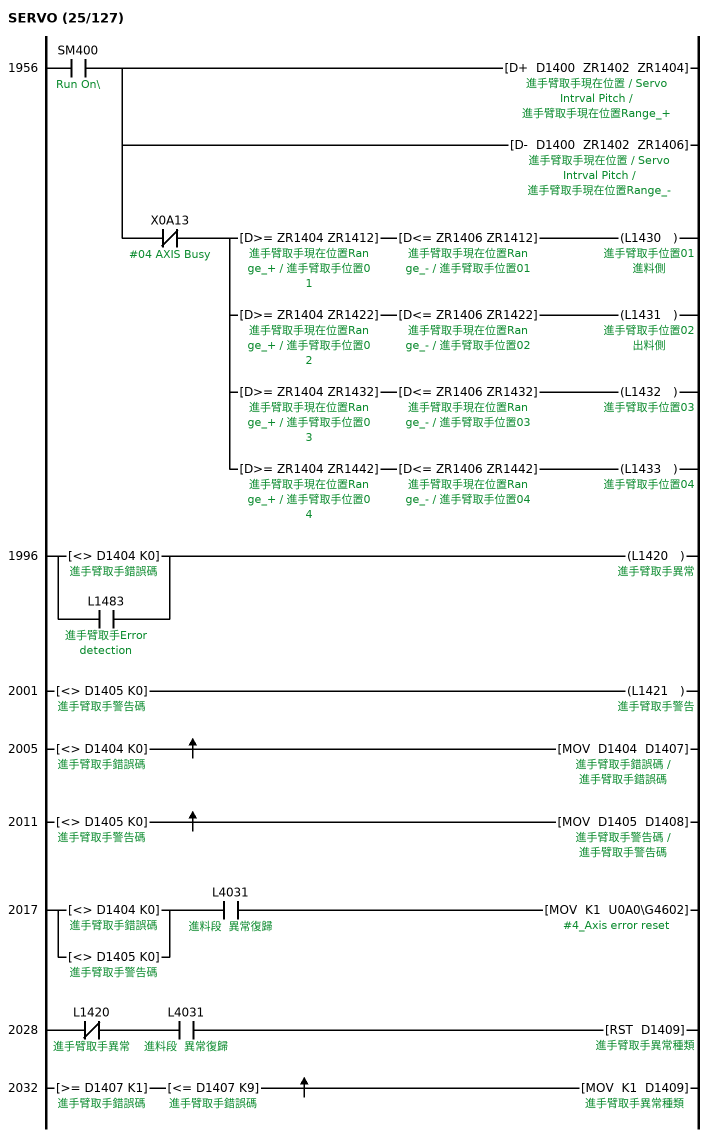
[picture p24: ladder of SERVO, rungs at steps 1956 to 2032]
1956  LD      SM400  ; Run On\
      D+      D1400 ZR1402 ZR1404  ; 進手臂取手現在位置Range_+
      D-      D1400 ZR1402 ZR1406  ; 進手臂取手現在位置Range_-
      ANI     X0A13  ; #04 AXIS Busy
      MPS
      ANDD>=  ZR1404 ZR1412  ; 進手臂取手現在位置Range_+ / 進手臂取手位置01
      ANDD<=  ZR1406 ZR1412  ; 進手臂取手現在位置Range_- / 進手臂取手位置01
      OUT     L1430  ; 進手臂取手位置01  進料側
      MRD
      ANDD>=  ZR1404 ZR1422  ; 進手臂取手現在位置Range_+ / 進手臂取手位置02
      ANDD<=  ZR1406 ZR1422  ; 進手臂取手現在位置Range_- / 進手臂取手位置02
      OUT     L1431  ; 進手臂取手位置02  出料側
      MRD
      ANDD>=  ZR1404 ZR1432  ; 進手臂取手現在位置Range_+ / 進手臂取手位置03
      ANDD<=  ZR1406 ZR1432  ; 進手臂取手現在位置Range_- / 進手臂取手位置03
      OUT     L1432  ; 進手臂取手位置03
      MPP
      ANDD>=  ZR1404 ZR1442  ; 進手臂取手現在位置Range_+ / 進手臂取手位置04
      ANDD<=  ZR1406 ZR1442  ; 進手臂取手現在位置Range_- / 進手臂取手位置04
      OUT     L1433  ; 進手臂取手位置04
1996  LD<>    D1404 K0  ; 進手臂取手錯誤碼
      OR      L1483  ; 進手臂取手Error detection
      OUT     L1420  ; 進手臂取手異常
2001  LD<>    D1405 K0  ; 進手臂取手警告碼
      OUT     L1421  ; 進手臂取手警告
2005  LD<>    D1404 K0  ; 進手臂取手錯誤碼
      MEP
      MOV     D1404 D1407  ; 進手臂取手錯誤碼
2011  LD<>    D1405 K0  ; 進手臂取手警告碼
      MEP
      MOV     D1405 D1408  ; 進手臂取手警告碼
2017  LD<>    D1404 K0  ; 進手臂取手錯誤碼
      OR<>    D1405 K0  ; 進手臂取手警告碼
      AND     L4031  ; 進料段  異常復歸
      MOV     K1 U0A0\G4602  ; #4_Axis error reset
2028  LDI     L1420  ; 進手臂取手異常
      AND     L4031  ; 進料段  異常復歸
      RST     D1409  ; 進手臂取手異常種類
2032  LD>=    D1407 K1  ; 進手臂取手錯誤碼
      AND<=   D1407 K9  ; 進手臂取手錯誤碼
      MEP
      MOV     K1 D1409
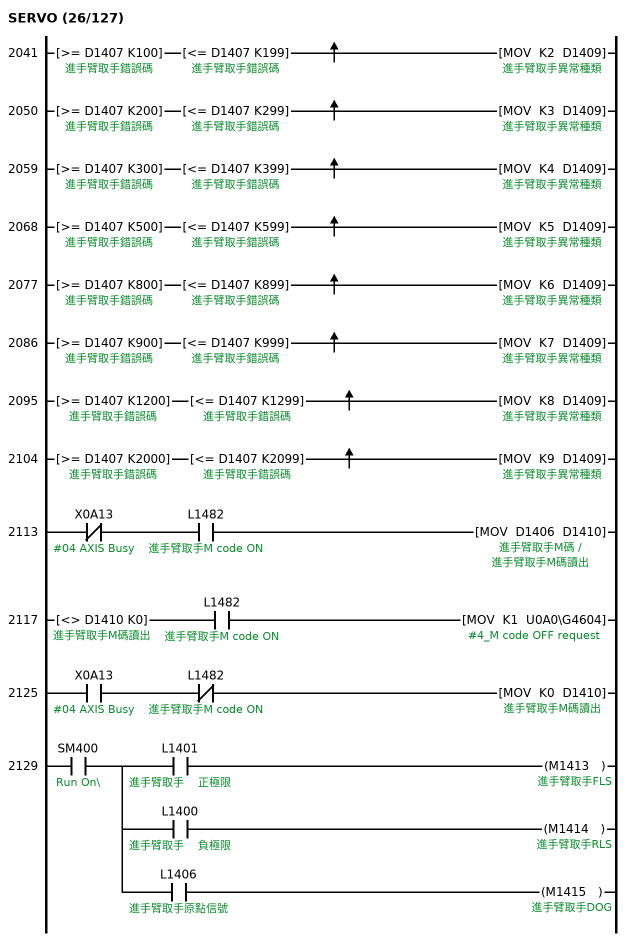
2041  LD>=    D1407 K100  ; 進手臂取手錯誤碼
      AND<=   D1407 K199  ; 進手臂取手錯誤碼
      MEP
      MOV     K2 D1409
2050  LD>=    D1407 K200  ; 進手臂取手錯誤碼
      AND<=   D1407 K299  ; 進手臂取手錯誤碼
      MEP
      MOV     K3 D1409
2059  LD>=    D1407 K300  ; 進手臂取手錯誤碼
      AND<=   D1407 K399  ; 進手臂取手錯誤碼
      MEP
      MOV     K4 D1409
2068  LD>=    D1407 K500  ; 進手臂取手錯誤碼
      AND<=   D1407 K599  ; 進手臂取手錯誤碼
      MEP
      MOV     K5 D1409
2077  LD>=    D1407 K800  ; 進手臂取手錯誤碼
      AND<=   D1407 K899  ; 進手臂取手錯誤碼
      MEP
      MOV     K6 D1409
2086  LD>=    D1407 K900  ; 進手臂取手錯誤碼
      AND<=   D1407 K999  ; 進手臂取手錯誤碼
      MEP
      MOV     K7 D1409
2095  LD>=    D1407 K1200  ; 進手臂取手錯誤碼
      AND<=   D1407 K1299  ; 進手臂取手錯誤碼
      MEP
      MOV     K8 D1409
2104  LD>=    D1407 K2000  ; 進手臂取手錯誤碼
      AND<=   D1407 K2099  ; 進手臂取手錯誤碼
      MEP
      MOV     K9 D1409
2113  LDI     X0A13  ; #04 AXIS Busy
      AND     L1482  ; 進手臂取手M code ON
      MOV     D1406 D1410  ; 進手臂取手M碼讀出
2117  LD<>    D1410 K0  ; 進手臂取手M碼讀出
      AND     L1482  ; 進手臂取手M code ON
      MOV     K1 U0A0\G4604  ; #4_M code OFF request
2125  LD      X0A13  ; #04 AXIS Busy
      ANI     L1482  ; 進手臂取手M code ON
      MOV     K0 D1410
2129  LD      SM400  ; Run On\
      MPS
      AND     L1401  ; 進手臂取手    正極限
      OUT     M1413  ; 進手臂取手FLS
      MRD
      AND     L1400  ; 進手臂取手    負極限
      OUT     M1414  ; 進手臂取手RLS
      MPP
      AND     L1406  ; 進手臂取手原點信號
      OUT     M1415  ; 進手臂取手DOG
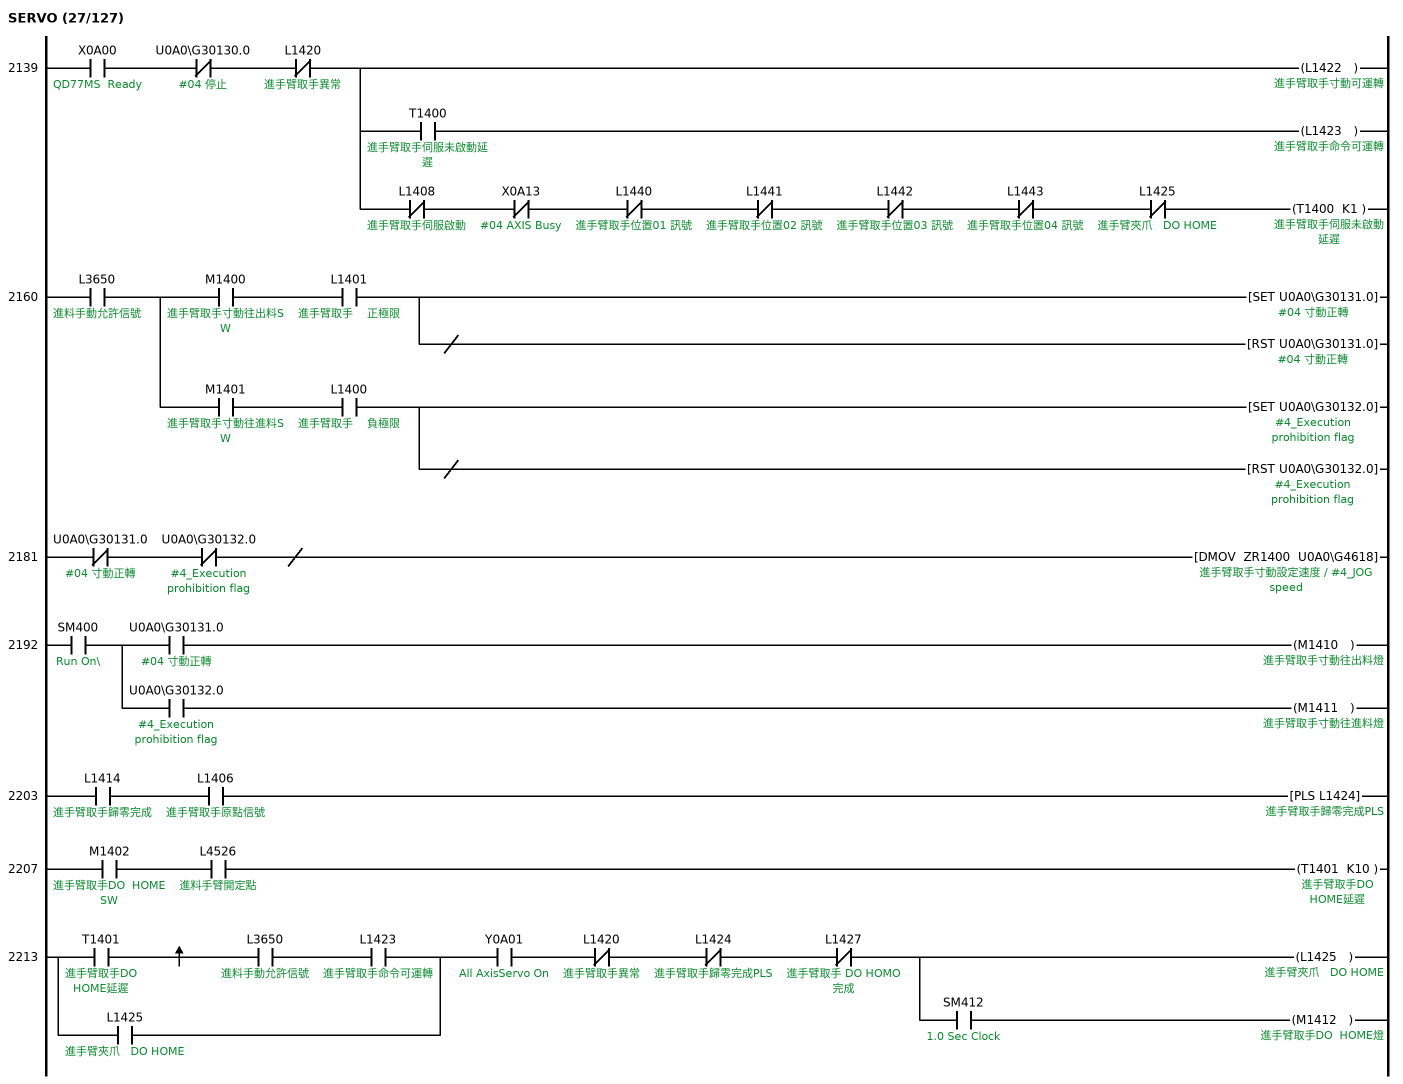
2139  LD      X0A00  ; QD77MS  Ready
      ANI     U0A0\G30130.0  ; #04 停止
      ANI     L1420  ; 進手臂取手異常
      OUT     L1422  ; 進手臂取手寸動可運轉
      MPS
      AND     T1400  ; 進手臂取手伺服未啟動延遲
      OUT     L1423  ; 進手臂取手命令可運轉
      MPP
      ANI     L1408  ; 進手臂取手伺服啟動
      ANI     X0A13  ; #04 AXIS Busy
      ANI     L1440  ; 進手臂取手位置01 訊號
      ANI     L1441  ; 進手臂取手位置02 訊號
      ANI     L1442  ; 進手臂取手位置03 訊號
      ANI     L1443  ; 進手臂取手位置04 訊號
      ANI     L1425  ; 進手臂夾爪   DO HOME
      OUT     T1400 K1  ; 進手臂取手伺服未啟動延遲
2160  LD      L3650  ; 進料手動允許信號
      MPS
      AND     M1400  ; 進手臂取手寸動往出料SW
      AND     L1401  ; 進手臂取手    正極限
      SET     U0A0\G30131.0  ; #04 寸動正轉
      INV
      RST     U0A0\G30131.0  ; #04 寸動正轉
      MPP
      AND     M1401  ; 進手臂取手寸動往進料SW
      AND     L1400  ; 進手臂取手    負極限
      SET     U0A0\G30132.0  ; #4_Execution prohibition flag
      INV
      RST     U0A0\G30132.0  ; #4_Execution prohibition flag
2181  LDI     U0A0\G30131.0  ; #04 寸動正轉
      ANI     U0A0\G30132.0  ; #4_Execution prohibition flag
      INV
      DMOV    ZR1400 U0A0\G4618  ; 進手臂取手寸動設定速度 / #4_JOG     speed
2192  LD      SM400  ; Run On\
      MPS
      AND     U0A0\G30131.0  ; #04 寸動正轉
      OUT     M1410  ; 進手臂取手寸動往出料燈
      MPP
      AND     U0A0\G30132.0  ; #4_Execution prohibition flag
      OUT     M1411  ; 進手臂取手寸動往進料燈
2203  LD      L1414  ; 進手臂取手歸零完成
      AND     L1406  ; 進手臂取手原點信號
      PLS     L1424  ; 進手臂取手歸零完成PLS
2207  LD      M1402  ; 進手臂取手DO  HOME SW
      AND     L4526  ; 進料手臂開定點
      OUT     T1401 K10  ; 進手臂取手DO HOME延遲
2213  LD      T1401  ; 進手臂取手DO HOME延遲
      MEP
      AND     L3650  ; 進料手動允許信號
      AND     L1423  ; 進手臂取手命令可運轉
      OR      L1425  ; 進手臂夾爪   DO HOME
      AND     Y0A01  ; All AxisServo On
      ANI     L1420  ; 進手臂取手異常
      ANI     L1424  ; 進手臂取手歸零完成PLS
      ANI     L1427  ; 進手臂取手 DO HOMO 完成
      OUT     L1425  ; 進手臂夾爪   DO HOME
      AND     SM412  ; 1.0 Sec Clock
      OUT     M1412  ; 進手臂取手DO  HOME燈
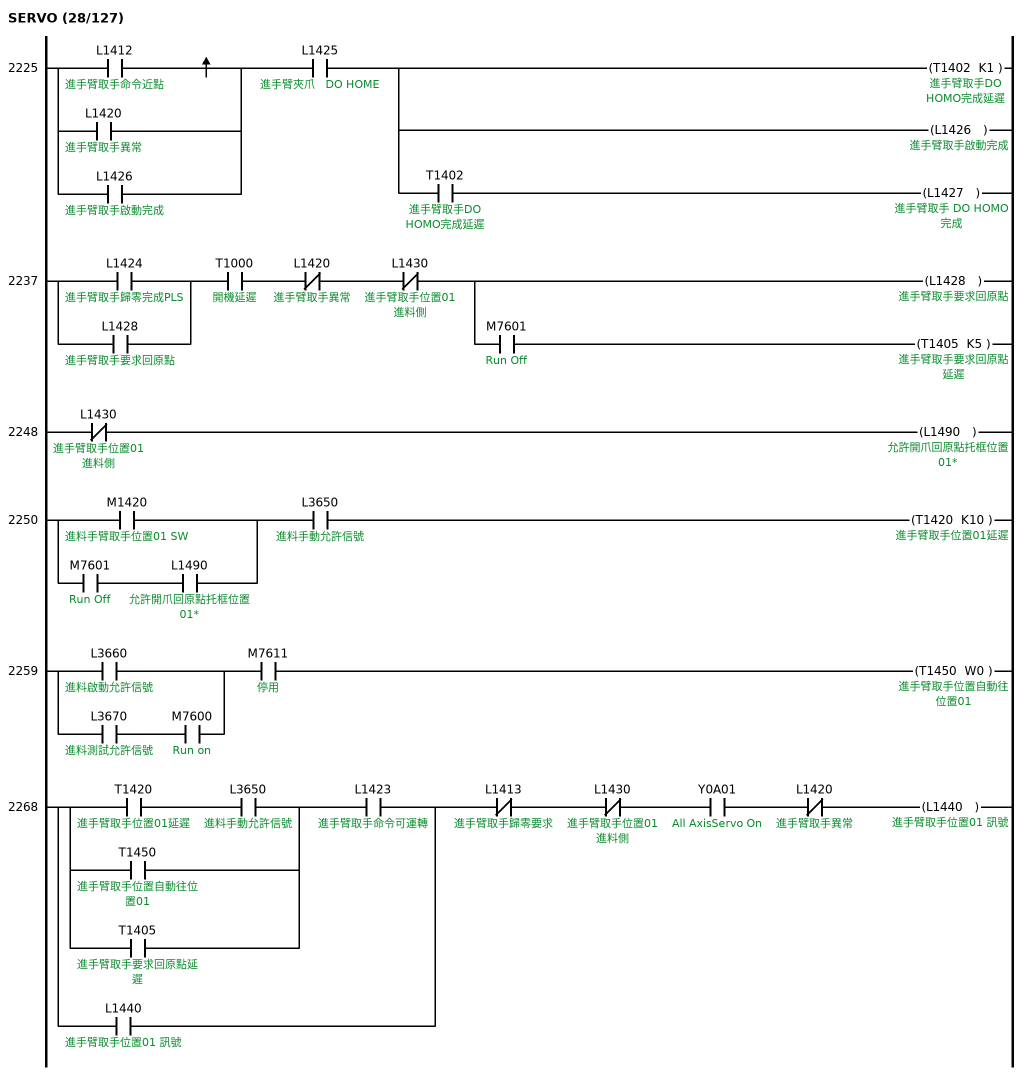
2225  LD      L1412  ; 進手臂取手命令近點
      MEP
      OR      L1420  ; 進手臂取手異常
      OR      L1426  ; 進手臂取手啟動完成
      AND     L1425  ; 進手臂夾爪   DO HOME
      OUT     T1402 K1  ; 進手臂取手DO HOMO完成延遲
      OUT     L1426  ; 進手臂取手啟動完成
      AND     T1402  ; 進手臂取手DO HOMO完成延遲
      OUT     L1427  ; 進手臂取手 DO HOMO 完成
2237  LD      L1424  ; 進手臂取手歸零完成PLS
      OR      L1428  ; 進手臂取手要求回原點
      AND     T1000  ; 開機延遲
      ANI     L1420  ; 進手臂取手異常
      ANI     L1430  ; 進手臂取手位置01  進料側
      OUT     L1428  ; 進手臂取手要求回原點
      AND     M7601  ; Run Off
      OUT     T1405 K5  ; 進手臂取手要求回原點延遲
2248  LDI     L1430  ; 進手臂取手位置01  進料側
      OUT     L1490  ; 允許開爪回原點托框位置01*
2250  LD      M1420  ; 進料手臂取手位置01 SW
      LD      M7601  ; Run Off
      AND     L1490  ; 允許開爪回原點托框位置01*
      ORB
      AND     L3650  ; 進料手動允許信號
      OUT     T1420 K10  ; 進手臂取手位置01延遲
2259  LD      L3660  ; 進料啟動允許信號
      LD      L3670  ; 進料測試允許信號
      AND     M7600  ; Run on
      ORB
      AND     M7611  ; 停用
      OUT     T1450 W0  ; 進手臂取手位置自動往位置01
2268  LD      T1420  ; 進手臂取手位置01延遲
      AND     L3650  ; 進料手動允許信號
      OR      T1450  ; 進手臂取手位置自動往位置01
      OR      T1405  ; 進手臂取手要求回原點延遲
      AND     L1423  ; 進手臂取手命令可運轉
      OR      L1440  ; 進手臂取手位置01 訊號
      ANI     L1413  ; 進手臂取手歸零要求
      ANI     L1430  ; 進手臂取手位置01  進料側
      AND     Y0A01  ; All AxisServo On
      ANI     L1420  ; 進手臂取手異常
      OUT     L1440  ; 進手臂取手位置01 訊號
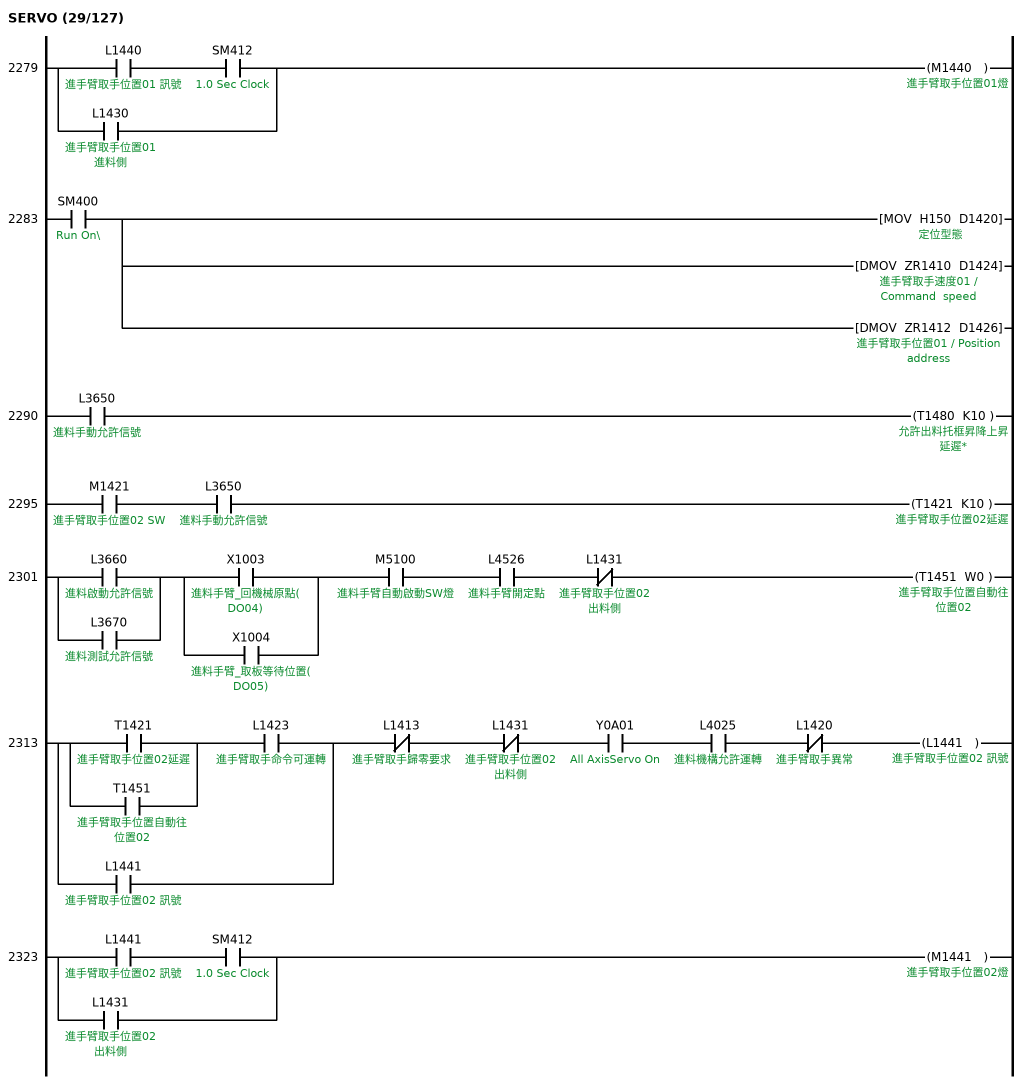
2279  LD      L1440  ; 進手臂取手位置01 訊號
      AND     SM412  ; 1.0 Sec Clock
      OR      L1430  ; 進手臂取手位置01  進料側
      OUT     M1440  ; 進手臂取手位置01燈
2283  LD      SM400  ; Run On\
      MOV     H150 D1420  ; 定位型態
      DMOV    ZR1410 D1424  ; 進手臂取手速度01 / Command  speed
      DMOV    ZR1412 D1426  ; Position address
2290  LD      L3650  ; 進料手動允許信號
      OUT     T1480 K10  ; 允許出料托框昇降上昇延遲*
2295  LD      M1421  ; 進手臂取手位置02 SW
      AND     L3650  ; 進料手動允許信號
      OUT     T1421 K10  ; 進手臂取手位置02延遲
2301  LD      L3660  ; 進料啟動允許信號
      OR      L3670  ; 進料測試允許信號
      LD      X1003  ; 進料手臂_回機械原點(DO04)
      OR      X1004  ; 進料手臂_取板等待位置(DO05)
      ANB
      AND     M5100  ; 進料手臂自動啟動SW燈
      AND     L4526  ; 進料手臂開定點
      ANI     L1431  ; 進手臂取手位置02  出料側
      OUT     T1451 W0  ; 進手臂取手位置自動往  位置02
2313  LD      T1421  ; 進手臂取手位置02延遲
      OR      T1451  ; 進手臂取手位置自動往  位置02
      AND     L1423  ; 進手臂取手命令可運轉
      OR      L1441  ; 進手臂取手位置02 訊號
      ANI     L1413  ; 進手臂取手歸零要求
      ANI     L1431  ; 進手臂取手位置02  出料側
      AND     Y0A01  ; All AxisServo On
      AND     L4025  ; 進料機構允許運轉
      ANI     L1420  ; 進手臂取手異常
      OUT     L1441  ; 進手臂取手位置02 訊號
2323  LD      L1441  ; 進手臂取手位置02 訊號
      AND     SM412  ; 1.0 Sec Clock
      OR      L1431  ; 進手臂取手位置02  出料側
      OUT     M1441  ; 進手臂取手位置02燈
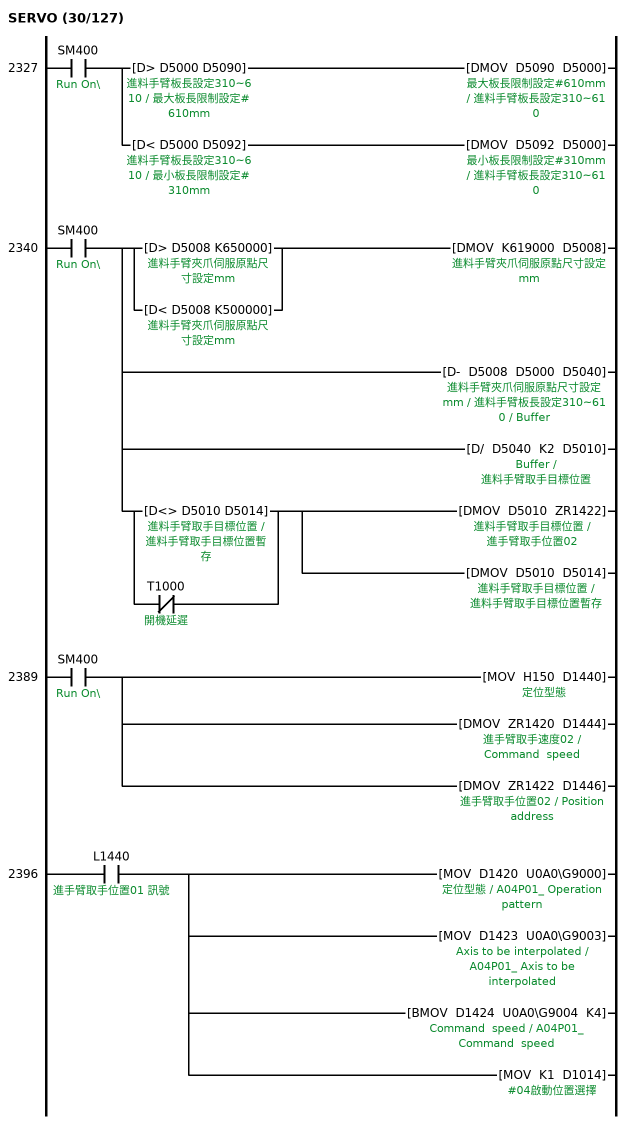
2327  LD      SM400  ; Run On\
      MPS
      ANDD>   D5000 D5090  ; 進料手臂板長設定310~610 / 最大板長限制設定#610mm
      DMOV    D5090 D5000
      MPP
      ANDD<   D5000 D5092  ; 進料手臂板長設定310~610 / 最小板長限制設定#310mm
      DMOV    D5092 D5000
2340  LD      SM400  ; Run On\
      MPS
      LDD>    D5008 K650000  ; 進料手臂夾爪伺服原點尺寸設定mm
      ORD<    D5008 K500000  ; 進料手臂夾爪伺服原點尺寸設定mm
      ANB
      DMOV    K619000 D5008
        [note] /* 手臂夾爪伺服原點尺寸_619mm */
      MPP
      D-      D5008 D5000 D5040
      D/      D5040 K2 D5010  ; 進料手臂取手目標位置
      LDD<>   D5010 D5014  ; 進料手臂取手目標位置 / 進料手臂取手目標位置暫存
      ORI     T1000  ; 開機延遲
      ANB
      DMOV    D5010 ZR1422
      DMOV    D5010 D5014
2389  LD      SM400  ; Run On\
      MOV     H150 D1440  ; 定位型態
      DMOV    ZR1420 D1444  ; 進手臂取手速度02 / Command  speed
      DMOV    ZR1422 D1446  ; Position address
2396  LD      L1440  ; 進手臂取手位置01 訊號
      MOV     D1420 U0A0\G9000  ; A04P01_ Operation pattern
      MOV     D1423 U0A0\G9003  ; Axis to be interpolated / A04P01_ Axis to be interpolated
      BMOV    D1424 U0A0\G9004 K4  ; A04P01_ Command  speed
      MOV     K1 D1014  ; #04啟動位置選擇
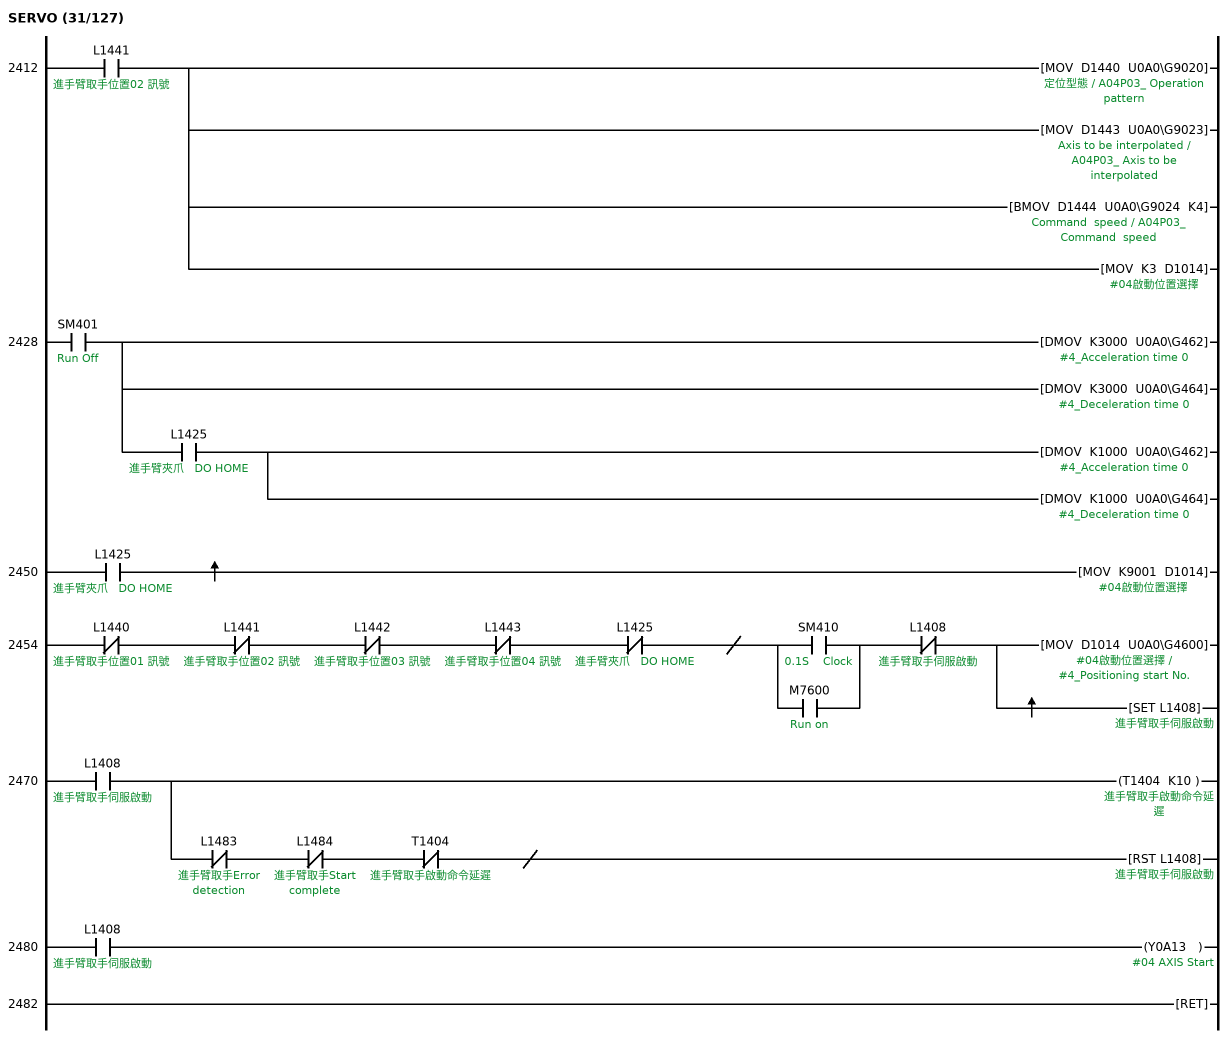
2412  LD      L1441  ; 進手臂取手位置02 訊號
      MOV     D1440 U0A0\G9020  ; A04P03_ Operation pattern
      MOV     D1443 U0A0\G9023  ; Axis to be interpolated / A04P03_ Axis to be interpolated
      BMOV    D1444 U0A0\G9024 K4  ; A04P03_ Command  speed
      MOV     K3 D1014
2428  LD      SM401  ; Run Off
      DMOV    K3000 U0A0\G462  ; #4_Acceleration time 0
      DMOV    K3000 U0A0\G464  ; #4_Deceleration time 0
      AND     L1425  ; 進手臂夾爪   DO HOME
      DMOV    K1000 U0A0\G462
      DMOV    K1000 U0A0\G464
2450  LD      L1425  ; 進手臂夾爪   DO HOME
      MEP
      MOV     K9001 D1014
2454  LDI     L1440  ; 進手臂取手位置01 訊號
      ANI     L1441  ; 進手臂取手位置02 訊號
      ANI     L1442  ; 進手臂取手位置03 訊號
      ANI     L1443  ; 進手臂取手位置04 訊號
      ANI     L1425  ; 進手臂夾爪   DO HOME
      INV
      LD      SM410  ; 0.1S    Clock
      OR      M7600  ; Run on
      ANB
      ANI     L1408  ; 進手臂取手伺服啟動
      MOV     D1014 U0A0\G4600  ; #4_Positioning start No.
      MEP
      SET     L1408  ; 進手臂取手伺服啟動
2470  LD      L1408  ; 進手臂取手伺服啟動
      OUT     T1404 K10  ; 進手臂取手啟動命令延遲
      ANI     L1483  ; 進手臂取手Error detection
      ANI     L1484  ; 進手臂取手Start complete
      ANI     T1404  ; 進手臂取手啟動命令延遲
      INV
      RST     L1408  ; 進手臂取手伺服啟動
2480  LD      L1408  ; 進手臂取手伺服啟動
      OUT     Y0A13  ; #04 AXIS Start
2482  RET
      P1500
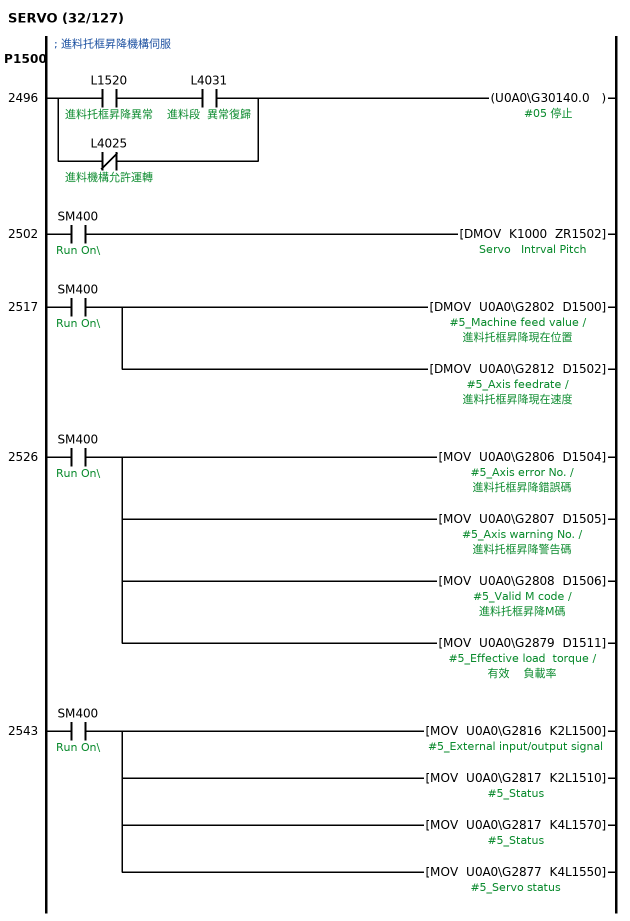
; 進料托框昇降機構伺服
2496  LD      L1520  ; 進料托框昇降異常
      AND     L4031  ; 進料段  異常復歸
      ORI     L4025  ; 進料機構允許運轉
      OUT     U0A0\G30140.0  ; #05 停止
2502  LD      SM400  ; Run On\
      DMOV    K1000 ZR1502  ; Servo   Intrval Pitch
        [note] /* Unit_1.000mm */
2517  LD      SM400  ; Run On\
      DMOV    U0A0\G2802 D1500  ; #5_Machine feed value / 進料托框昇降現在位置
      DMOV    U0A0\G2812 D1502  ; #5_Axis feedrate / 進料托框昇降現在速度
2526  LD      SM400  ; Run On\
      MOV     U0A0\G2806 D1504  ; #5_Axis error No. / 進料托框昇降錯誤碼
      MOV     U0A0\G2807 D1505  ; #5_Axis warning No. / 進料托框昇降警告碼
      MOV     U0A0\G2808 D1506  ; #5_Valid M code / 進料托框昇降M碼
      MOV     U0A0\G2879 D1511  ; #5_Effective load  torque / 有效    負載率
2543  LD      SM400  ; Run On\
      MOV     U0A0\G2816 K2L1500  ; #5_External input/output signal / 進料托框昇降   負極限
      MOV     U0A0\G2817 K2L1510  ; #5_Status / 進料托框昇降速度控制
      MOV     U0A0\G2817 K4L1570  ; 進料托框昇降速度控制
      MOV     U0A0\G2877 K4L1550  ; #5_Servo status / READY ON
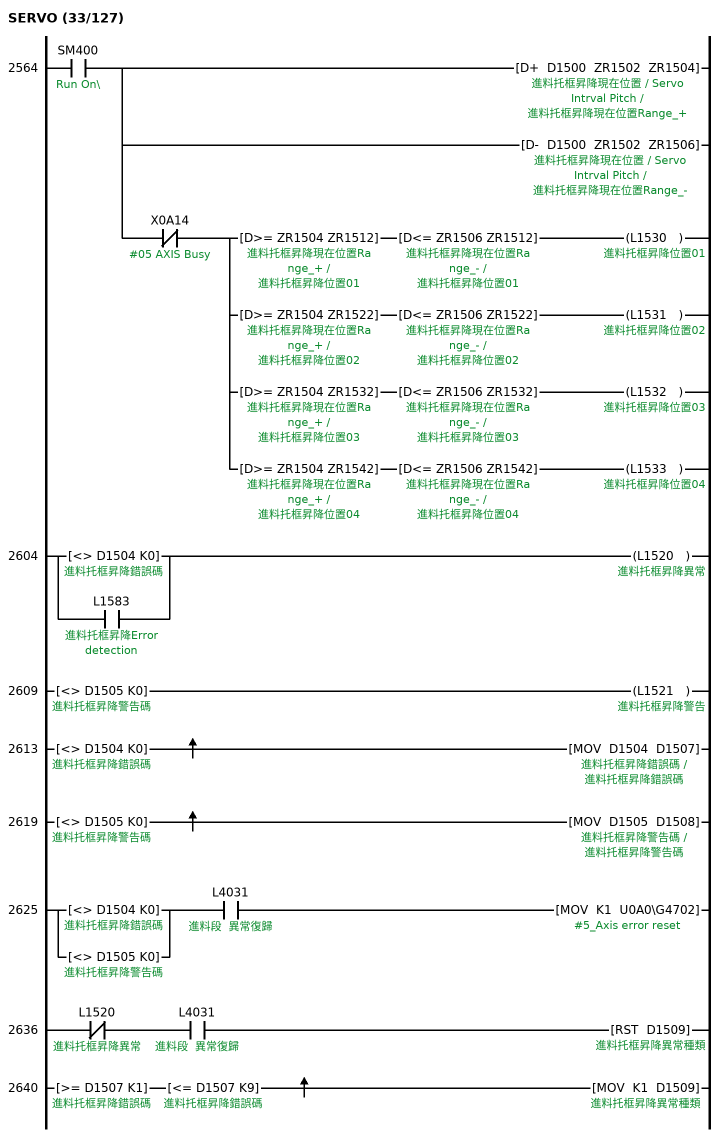
2564  LD      SM400  ; Run On\
      D+      D1500 ZR1502 ZR1504  ; 進料托框昇降現在位置Range_+
      D-      D1500 ZR1502 ZR1506  ; 進料托框昇降現在位置Range_-
      ANI     X0A14  ; #05 AXIS Busy
      MPS
      ANDD>=  ZR1504 ZR1512  ; 進料托框昇降現在位置Range_+ / 進料托框昇降位置01
      ANDD<=  ZR1506 ZR1512  ; 進料托框昇降現在位置Range_- / 進料托框昇降位置01
      OUT     L1530  ; 進料托框昇降位置01
      MRD
      ANDD>=  ZR1504 ZR1522  ; 進料托框昇降現在位置Range_+ / 進料托框昇降位置02
      ANDD<=  ZR1506 ZR1522  ; 進料托框昇降現在位置Range_- / 進料托框昇降位置02
      OUT     L1531  ; 進料托框昇降位置02
      MRD
      ANDD>=  ZR1504 ZR1532  ; 進料托框昇降現在位置Range_+ / 進料托框昇降位置03
      ANDD<=  ZR1506 ZR1532  ; 進料托框昇降現在位置Range_- / 進料托框昇降位置03
      OUT     L1532  ; 進料托框昇降位置03
      MPP
      ANDD>=  ZR1504 ZR1542  ; 進料托框昇降現在位置Range_+ / 進料托框昇降位置04
      ANDD<=  ZR1506 ZR1542  ; 進料托框昇降現在位置Range_- / 進料托框昇降位置04
      OUT     L1533  ; 進料托框昇降位置04
2604  LD<>    D1504 K0  ; 進料托框昇降錯誤碼
      OR      L1583  ; 進料托框昇降Error detection
      OUT     L1520  ; 進料托框昇降異常
2609  LD<>    D1505 K0  ; 進料托框昇降警告碼
      OUT     L1521  ; 進料托框昇降警告
2613  LD<>    D1504 K0  ; 進料托框昇降錯誤碼
      MEP
      MOV     D1504 D1507  ; 進料托框昇降錯誤碼
2619  LD<>    D1505 K0  ; 進料托框昇降警告碼
      MEP
      MOV     D1505 D1508  ; 進料托框昇降警告碼
2625  LD<>    D1504 K0  ; 進料托框昇降錯誤碼
      OR<>    D1505 K0  ; 進料托框昇降警告碼
      AND     L4031  ; 進料段  異常復歸
      MOV     K1 U0A0\G4702  ; #5_Axis error reset
2636  LDI     L1520  ; 進料托框昇降異常
      AND     L4031  ; 進料段  異常復歸
      RST     D1509  ; 進料托框昇降異常種類
2640  LD>=    D1507 K1  ; 進料托框昇降錯誤碼
      AND<=   D1507 K9  ; 進料托框昇降錯誤碼
      MEP
      MOV     K1 D1509
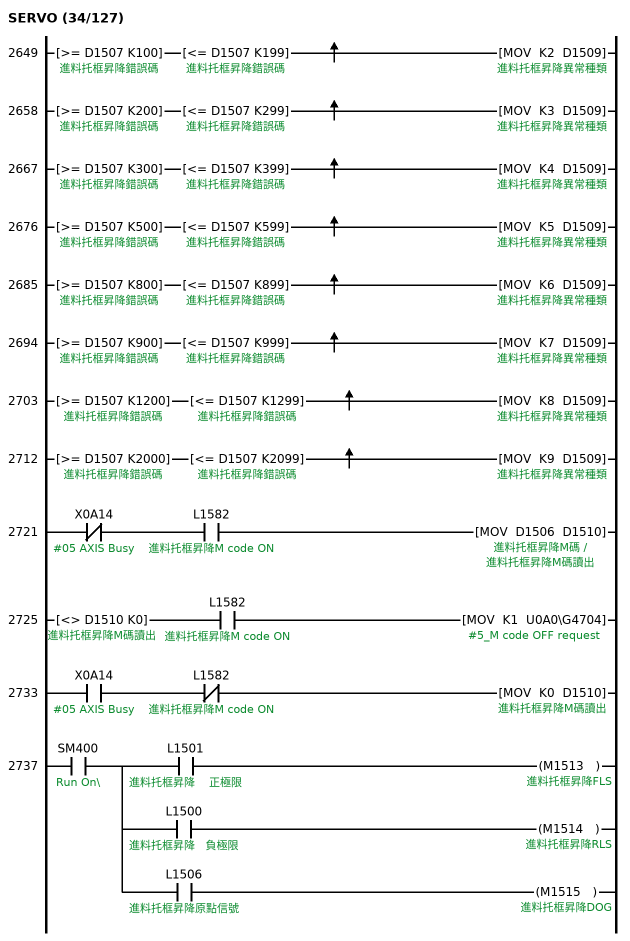
2649  LD>=    D1507 K100  ; 進料托框昇降錯誤碼
      AND<=   D1507 K199  ; 進料托框昇降錯誤碼
      MEP
      MOV     K2 D1509
2658  LD>=    D1507 K200  ; 進料托框昇降錯誤碼
      AND<=   D1507 K299  ; 進料托框昇降錯誤碼
      MEP
      MOV     K3 D1509
2667  LD>=    D1507 K300  ; 進料托框昇降錯誤碼
      AND<=   D1507 K399  ; 進料托框昇降錯誤碼
      MEP
      MOV     K4 D1509
2676  LD>=    D1507 K500  ; 進料托框昇降錯誤碼
      AND<=   D1507 K599  ; 進料托框昇降錯誤碼
      MEP
      MOV     K5 D1509
2685  LD>=    D1507 K800  ; 進料托框昇降錯誤碼
      AND<=   D1507 K899  ; 進料托框昇降錯誤碼
      MEP
      MOV     K6 D1509
2694  LD>=    D1507 K900  ; 進料托框昇降錯誤碼
      AND<=   D1507 K999  ; 進料托框昇降錯誤碼
      MEP
      MOV     K7 D1509
2703  LD>=    D1507 K1200  ; 進料托框昇降錯誤碼
      AND<=   D1507 K1299  ; 進料托框昇降錯誤碼
      MEP
      MOV     K8 D1509
2712  LD>=    D1507 K2000  ; 進料托框昇降錯誤碼
      AND<=   D1507 K2099  ; 進料托框昇降錯誤碼
      MEP
      MOV     K9 D1509
2721  LDI     X0A14  ; #05 AXIS Busy
      AND     L1582  ; 進料托框昇降M code ON
      MOV     D1506 D1510  ; 進料托框昇降M碼讀出
2725  LD<>    D1510 K0  ; 進料托框昇降M碼讀出
      AND     L1582  ; 進料托框昇降M code ON
      MOV     K1 U0A0\G4704  ; #5_M code OFF request
2733  LD      X0A14  ; #05 AXIS Busy
      ANI     L1582  ; 進料托框昇降M code ON
      MOV     K0 D1510
2737  LD      SM400  ; Run On\
      MPS
      AND     L1501  ; 進料托框昇降    正極限
      OUT     M1513  ; 進料托框昇降FLS
      MRD
      AND     L1500  ; 進料托框昇降   負極限
      OUT     M1514  ; 進料托框昇降RLS
      MPP
      AND     L1506  ; 進料托框昇降原點信號
      OUT     M1515  ; 進料托框昇降DOG
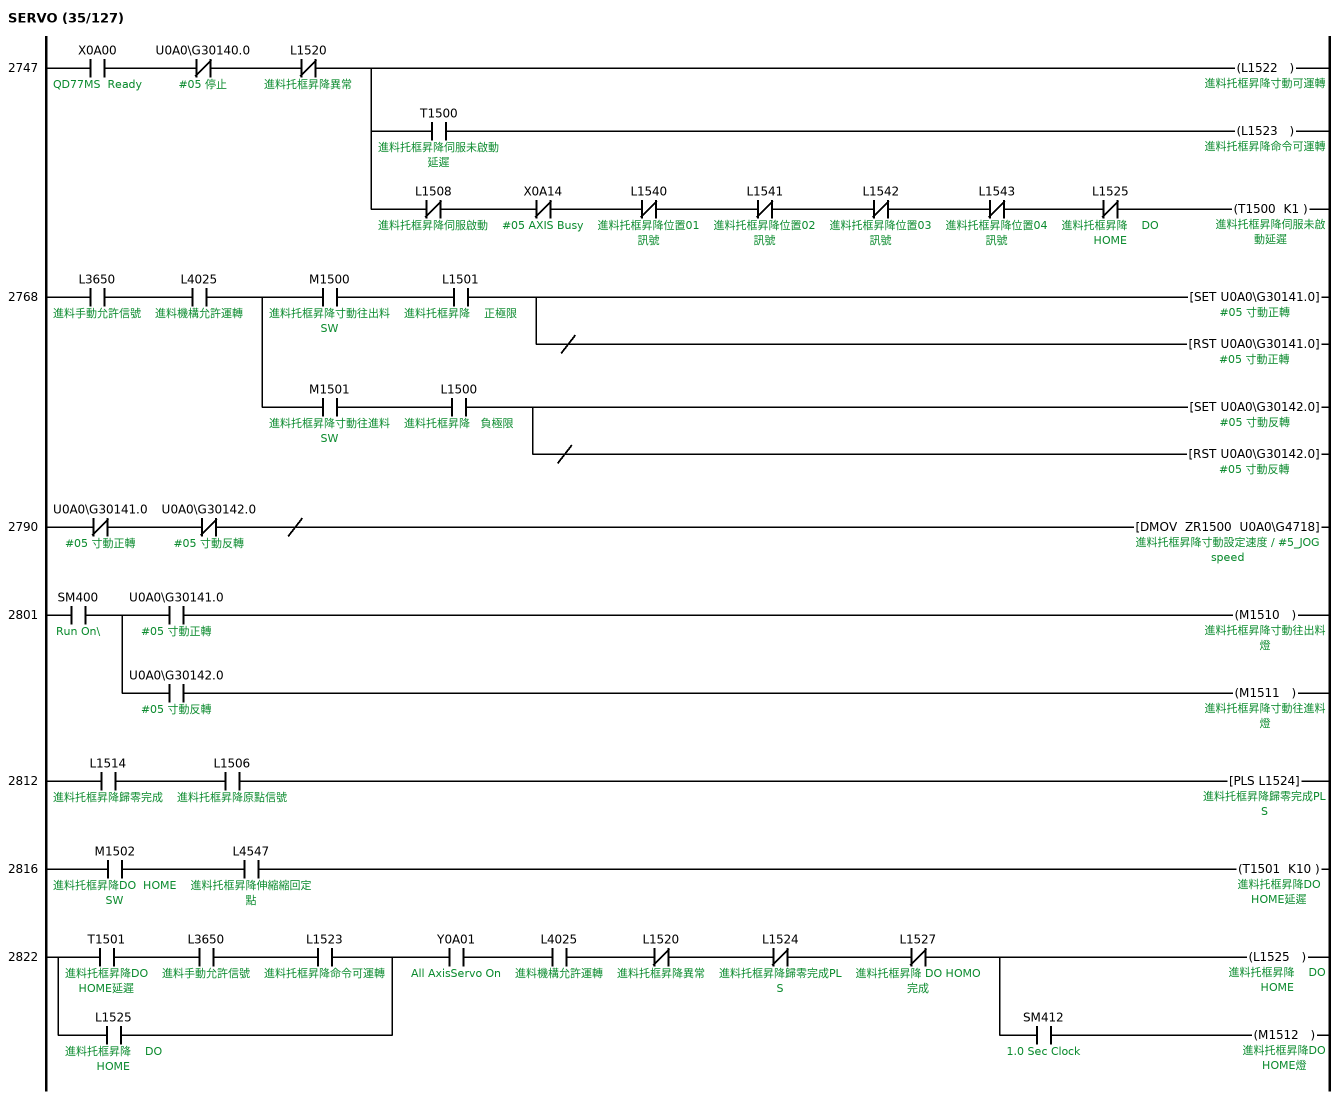
2747  LD      X0A00  ; QD77MS  Ready
      ANI     U0A0\G30140.0  ; #05 停止
      ANI     L1520  ; 進料托框昇降異常
      OUT     L1522  ; 進料托框昇降寸動可運轉
      MPS
      AND     T1500  ; 進料托框昇降伺服未啟動延遲
      OUT     L1523  ; 進料托框昇降命令可運轉
      MPP
      ANI     L1508  ; 進料托框昇降伺服啟動
      ANI     X0A14  ; #05 AXIS Busy
      ANI     L1540  ; 進料托框昇降位置01 訊號
      ANI     L1541  ; 進料托框昇降位置02 訊號
      ANI     L1542  ; 進料托框昇降位置03 訊號
      ANI     L1543  ; 進料托框昇降位置04 訊號
      ANI     L1525  ; 進料托框昇降    DO HOME
      OUT     T1500 K1  ; 進料托框昇降伺服未啟動延遲
2768  LD      L3650  ; 進料手動允許信號
      AND     L4025  ; 進料機構允許運轉
      MPS
      AND     M1500  ; 進料托框昇降寸動往出料SW
      AND     L1501  ; 進料托框昇降    正極限
      SET     U0A0\G30141.0  ; #05 寸動正轉
      INV
      RST     U0A0\G30141.0  ; #05 寸動正轉
      MPP
      AND     M1501  ; 進料托框昇降寸動往進料SW
      AND     L1500  ; 進料托框昇降   負極限
      SET     U0A0\G30142.0  ; #05 寸動反轉
      INV
      RST     U0A0\G30142.0  ; #05 寸動反轉
2790  LDI     U0A0\G30141.0  ; #05 寸動正轉
      ANI     U0A0\G30142.0  ; #05 寸動反轉
      INV
      DMOV    ZR1500 U0A0\G4718  ; 進料托框昇降寸動設定速度 / #5_JOG     speed
2801  LD      SM400  ; Run On\
      MPS
      AND     U0A0\G30141.0  ; #05 寸動正轉
      OUT     M1510  ; 進料托框昇降寸動往出料燈
      MPP
      AND     U0A0\G30142.0  ; #05 寸動反轉
      OUT     M1511  ; 進料托框昇降寸動往進料燈
2812  LD      L1514  ; 進料托框昇降歸零完成
      AND     L1506  ; 進料托框昇降原點信號
      PLS     L1524  ; 進料托框昇降歸零完成PLS
2816  LD      M1502  ; 進料托框昇降DO  HOME SW
      AND     L4547  ; 進料托框昇降伸縮縮回定點
      OUT     T1501 K10  ; 進料托框昇降DO HOME延遲
2822  LD      T1501  ; 進料托框昇降DO HOME延遲
      AND     L3650  ; 進料手動允許信號
      AND     L1523  ; 進料托框昇降命令可運轉
      OR      L1525  ; 進料托框昇降    DO HOME
      AND     Y0A01  ; All AxisServo On
      AND     L4025  ; 進料機構允許運轉
      ANI     L1520  ; 進料托框昇降異常
      ANI     L1524  ; 進料托框昇降歸零完成PLS
      ANI     L1527  ; 進料托框昇降 DO HOMO 完成
      OUT     L1525  ; 進料托框昇降    DO HOME
      AND     SM412  ; 1.0 Sec Clock
      OUT     M1512  ; 進料托框昇降DO  HOME燈
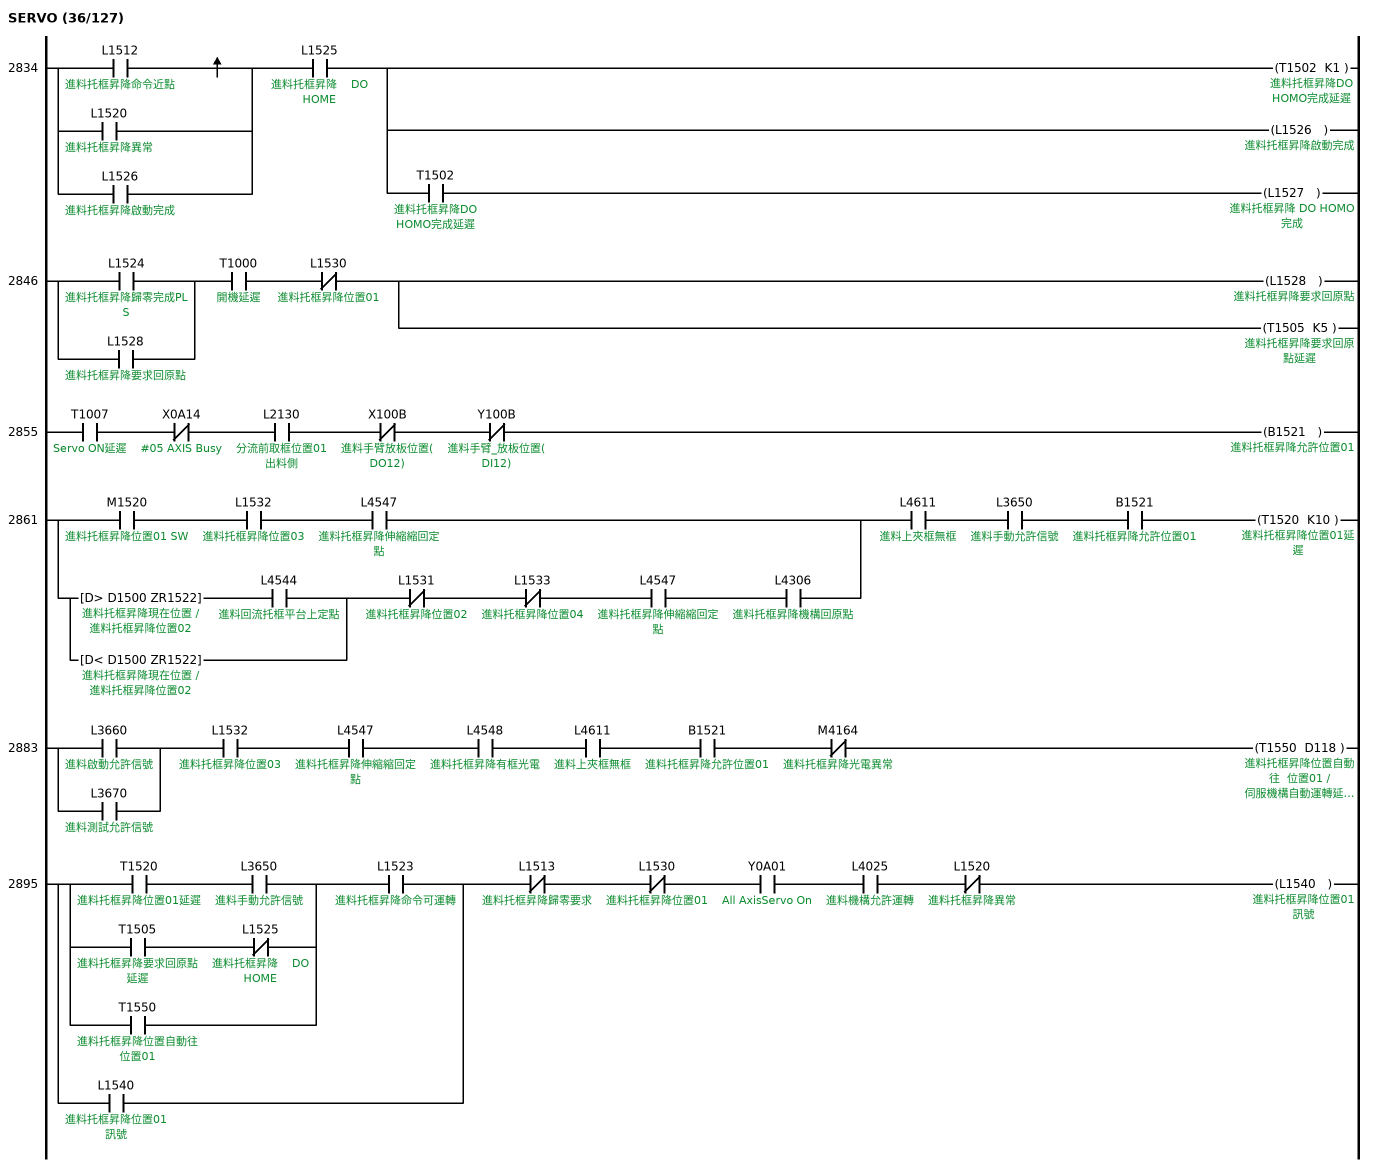
2834  LD      L1512  ; 進料托框昇降命令近點
      MEP
      OR      L1520  ; 進料托框昇降異常
      OR      L1526  ; 進料托框昇降啟動完成
      AND     L1525  ; 進料托框昇降    DO HOME
      OUT     T1502 K1  ; 進料托框昇降DO HOMO完成延遲
      OUT     L1526  ; 進料托框昇降啟動完成
      AND     T1502  ; 進料托框昇降DO HOMO完成延遲
      OUT     L1527  ; 進料托框昇降 DO HOMO 完成
2846  LD      L1524  ; 進料托框昇降歸零完成PLS
      OR      L1528  ; 進料托框昇降要求回原點
      AND     T1000  ; 開機延遲
      ANI     L1530  ; 進料托框昇降位置01
      OUT     L1528  ; 進料托框昇降要求回原點
      OUT     T1505 K5  ; 進料托框昇降要求回原點延遲
2855  LD      T1007  ; Servo ON延遲
      ANI     X0A14  ; #05 AXIS Busy
      AND     L2130  ; 分流前取框位置01  出料側
      ANI     X100B  ; 進料手臂放板位置(DO12)
      ANI     Y100B  ; 進料手臂_放板位置(DI12)
      OUT     B1521  ; 進料托框昇降允許位置01
2861  LD      M1520  ; 進料托框昇降位置01 SW
      AND     L1532  ; 進料托框昇降位置03
      AND     L4547  ; 進料托框昇降伸縮縮回定點
      LDD>    D1500 ZR1522  ; 進料托框昇降現在位置 / 進料托框昇降位置02
      AND     L4544  ; 進料回流托框平台上定點
      ORD<    D1500 ZR1522  ; 進料托框昇降現在位置 / 進料托框昇降位置02
      ANI     L1531  ; 進料托框昇降位置02
      ANI     L1533  ; 進料托框昇降位置04
      AND     L4547  ; 進料托框昇降伸縮縮回定點
      AND     L4306  ; 進料托框昇降機構回原點
      ORB
      AND     L4611  ; 進料上夾框無框
      AND     L3650  ; 進料手動允許信號
      AND     B1521  ; 進料托框昇降允許位置01
      OUT     T1520 K10  ; 進料托框昇降位置01延遲
2883  LD      L3660  ; 進料啟動允許信號
      OR      L3670  ; 進料測試允許信號
      AND     L1532  ; 進料托框昇降位置03
      AND     L4547  ; 進料托框昇降伸縮縮回定點
      AND     L4548  ; 進料托框昇降有框光電
      AND     L4611  ; 進料上夾框無框
      AND     B1521  ; 進料托框昇降允許位置01
      ANI     M4164  ; 進料托框昇降光電異常
      OUT     T1550 D118  ; 進料托框昇降位置自動往  位置01 / 伺服機構自動運轉延遲時間
2895  LD      T1520  ; 進料托框昇降位置01延遲
      AND     L3650  ; 進料手動允許信號
      LD      T1505  ; 進料托框昇降要求回原點延遲
      ANI     L1525  ; 進料托框昇降    DO HOME
      ORB
      OR      T1550  ; 進料托框昇降位置自動往  位置01
      AND     L1523  ; 進料托框昇降命令可運轉
      OR      L1540  ; 進料托框昇降位置01 訊號
      ANI     L1513  ; 進料托框昇降歸零要求
      ANI     L1530  ; 進料托框昇降位置01
      AND     Y0A01  ; All AxisServo On
      AND     L4025  ; 進料機構允許運轉
      ANI     L1520  ; 進料托框昇降異常
      OUT     L1540  ; 進料托框昇降位置01 訊號
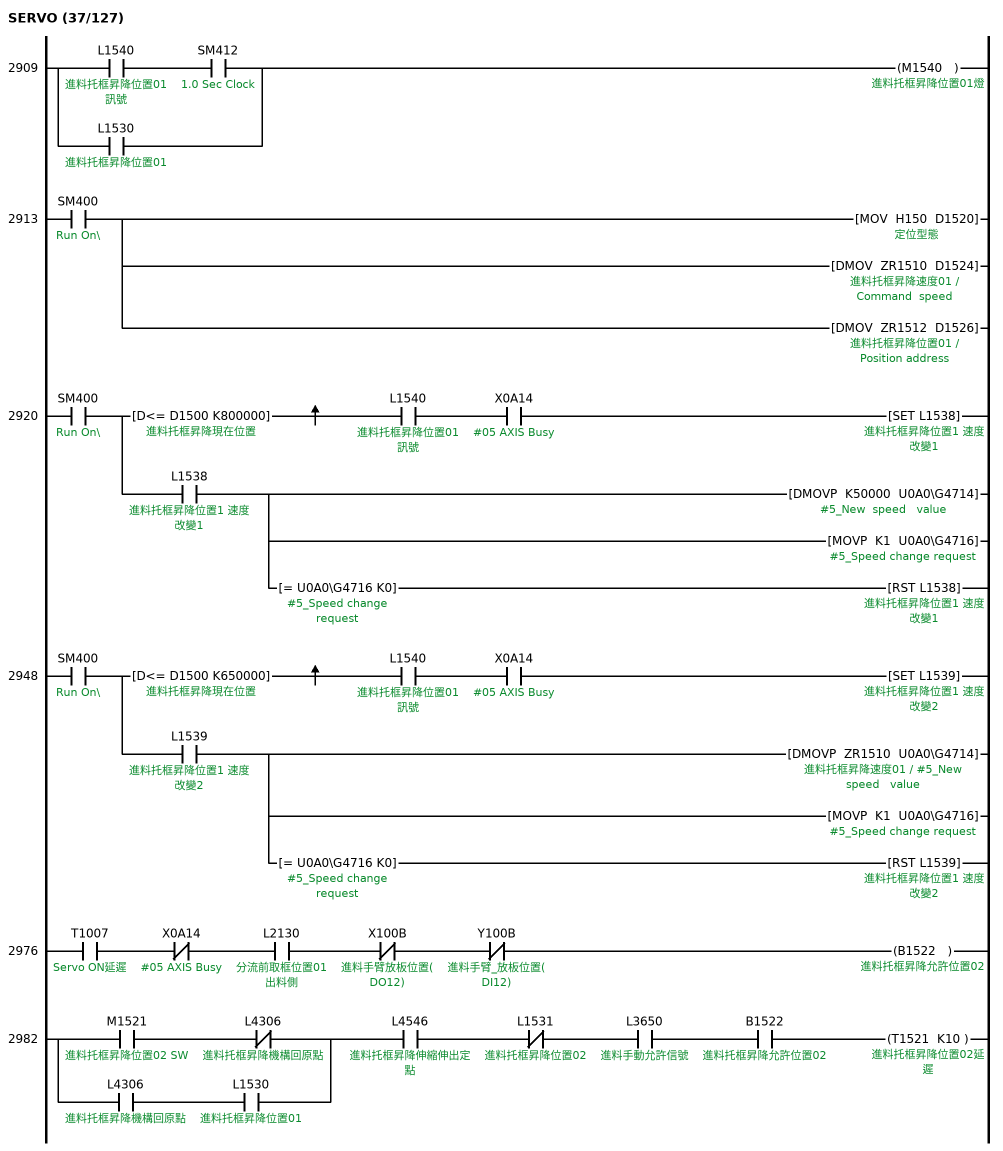
2909  LD      L1540  ; 進料托框昇降位置01 訊號
      AND     SM412  ; 1.0 Sec Clock
      OR      L1530  ; 進料托框昇降位置01
      OUT     M1540  ; 進料托框昇降位置01燈
2913  LD      SM400  ; Run On\
      MOV     H150 D1520  ; 定位型態
      DMOV    ZR1510 D1524  ; 進料托框昇降速度01 / Command  speed
      DMOV    ZR1512 D1526  ; Position address
2920  LD      SM400  ; Run On\
      MPS
      ANDD<=  D1500 K800000  ; 進料托框昇降現在位置
      MEP
      AND     L1540  ; 進料托框昇降位置01 訊號
      AND     X0A14  ; #05 AXIS Busy
      SET     L1538  ; 進料托框昇降位置1 速度  改變1
      MPP
      AND     L1538  ; 進料托框昇降位置1 速度  改變1
      DMOVP   K50000 U0A0\G4714  ; #5_New  speed   value
      MOVP    K1 U0A0\G4716  ; #5_Speed change request
      AND=    U0A0\G4716 K0  ; #5_Speed change request
      RST     L1538  ; 進料托框昇降位置1 速度  改變1
2948  LD      SM400  ; Run On\
      MPS
      ANDD<=  D1500 K650000  ; 進料托框昇降現在位置
      MEP
      AND     L1540  ; 進料托框昇降位置01 訊號
      AND     X0A14  ; #05 AXIS Busy
      SET     L1539  ; 進料托框昇降位置1 速度  改變2
      MPP
      AND     L1539  ; 進料托框昇降位置1 速度  改變2
      DMOVP   ZR1510 U0A0\G4714
      MOVP    K1 U0A0\G4716
      AND=    U0A0\G4716 K0  ; #5_Speed change request
      RST     L1539  ; 進料托框昇降位置1 速度  改變2
2976  LD      T1007  ; Servo ON延遲
      ANI     X0A14  ; #05 AXIS Busy
      AND     L2130  ; 分流前取框位置01  出料側
      ANI     X100B  ; 進料手臂放板位置(DO12)
      ANI     Y100B  ; 進料手臂_放板位置(DI12)
      OUT     B1522  ; 進料托框昇降允許位置02
2982  LD      M1521  ; 進料托框昇降位置02 SW
      ANI     L4306  ; 進料托框昇降機構回原點
      LD      L4306  ; 進料托框昇降機構回原點
      AND     L1530  ; 進料托框昇降位置01
      ORB
      AND     L4546  ; 進料托框昇降伸縮伸出定點
      ANI     L1531  ; 進料托框昇降位置02
      AND     L3650  ; 進料手動允許信號
      AND     B1522  ; 進料托框昇降允許位置02
      OUT     T1521 K10  ; 進料托框昇降位置02延遲
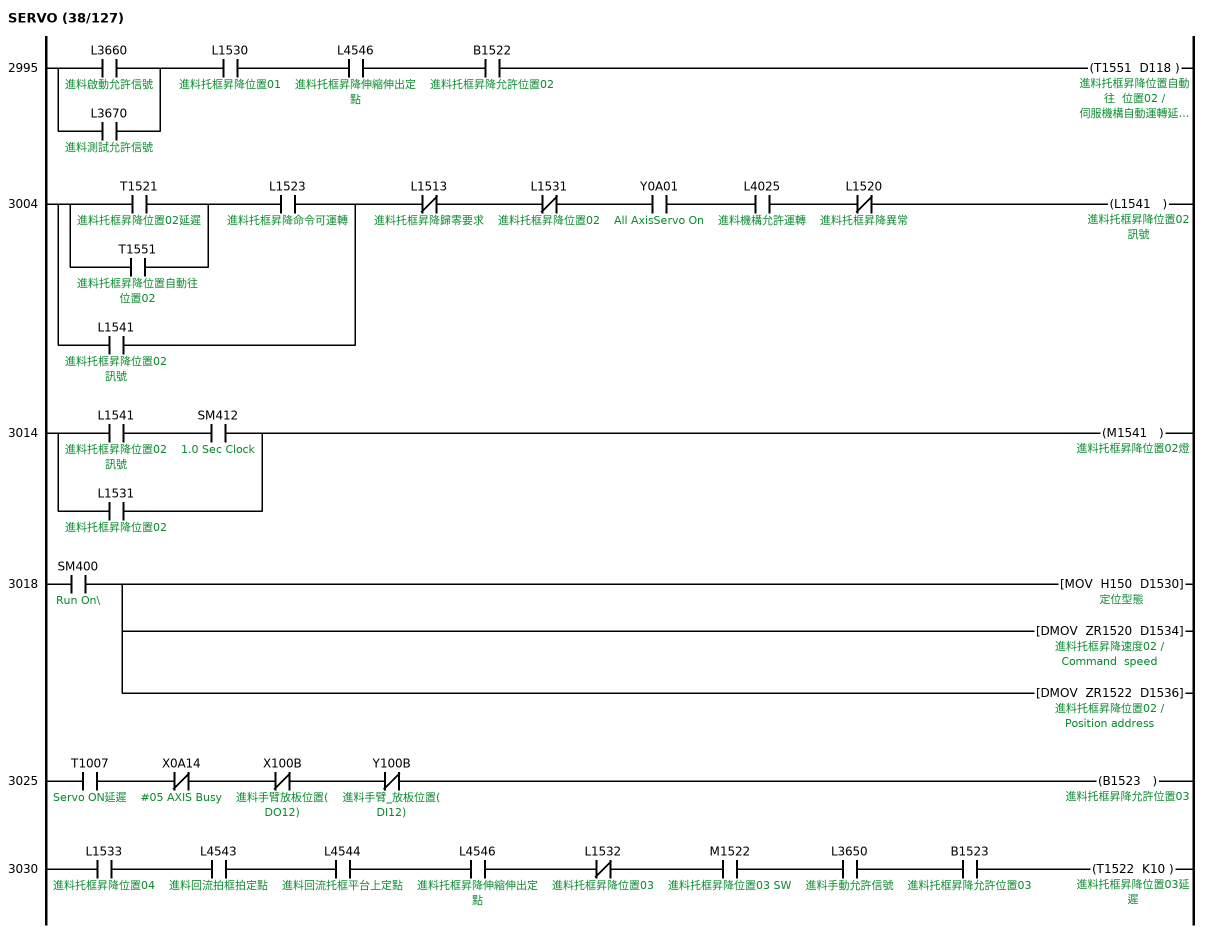
2995  LD      L3660  ; 進料啟動允許信號
      OR      L3670  ; 進料測試允許信號
      AND     L1530  ; 進料托框昇降位置01
      AND     L4546  ; 進料托框昇降伸縮伸出定點
      AND     B1522  ; 進料托框昇降允許位置02
      OUT     T1551 D118  ; 進料托框昇降位置自動往  位置02 / 伺服機構自動運轉延遲時間
3004  LD      T1521  ; 進料托框昇降位置02延遲
      OR      T1551  ; 進料托框昇降位置自動往  位置02
      AND     L1523  ; 進料托框昇降命令可運轉
      OR      L1541  ; 進料托框昇降位置02 訊號
      ANI     L1513  ; 進料托框昇降歸零要求
      ANI     L1531  ; 進料托框昇降位置02
      AND     Y0A01  ; All AxisServo On
      AND     L4025  ; 進料機構允許運轉
      ANI     L1520  ; 進料托框昇降異常
      OUT     L1541  ; 進料托框昇降位置02 訊號
3014  LD      L1541  ; 進料托框昇降位置02 訊號
      AND     SM412  ; 1.0 Sec Clock
      OR      L1531  ; 進料托框昇降位置02
      OUT     M1541  ; 進料托框昇降位置02燈
3018  LD      SM400  ; Run On\
      MOV     H150 D1530  ; 定位型態
      DMOV    ZR1520 D1534  ; 進料托框昇降速度02 / Command  speed
      DMOV    ZR1522 D1536  ; Position address
3025  LD      T1007  ; Servo ON延遲
      ANI     X0A14  ; #05 AXIS Busy
      ANI     X100B  ; 進料手臂放板位置(DO12)
      ANI     Y100B  ; 進料手臂_放板位置(DI12)
      OUT     B1523  ; 進料托框昇降允許位置03
3030  LD      L1533  ; 進料托框昇降位置04
      AND     L4543  ; 進料回流拍框拍定點
      AND     L4544  ; 進料回流托框平台上定點
      AND     L4546  ; 進料托框昇降伸縮伸出定點
      ANI     L1532  ; 進料托框昇降位置03
      AND     M1522  ; 進料托框昇降位置03 SW
      AND     L3650  ; 進料手動允許信號
      AND     B1523  ; 進料托框昇降允許位置03
      OUT     T1522 K10  ; 進料托框昇降位置03延遲
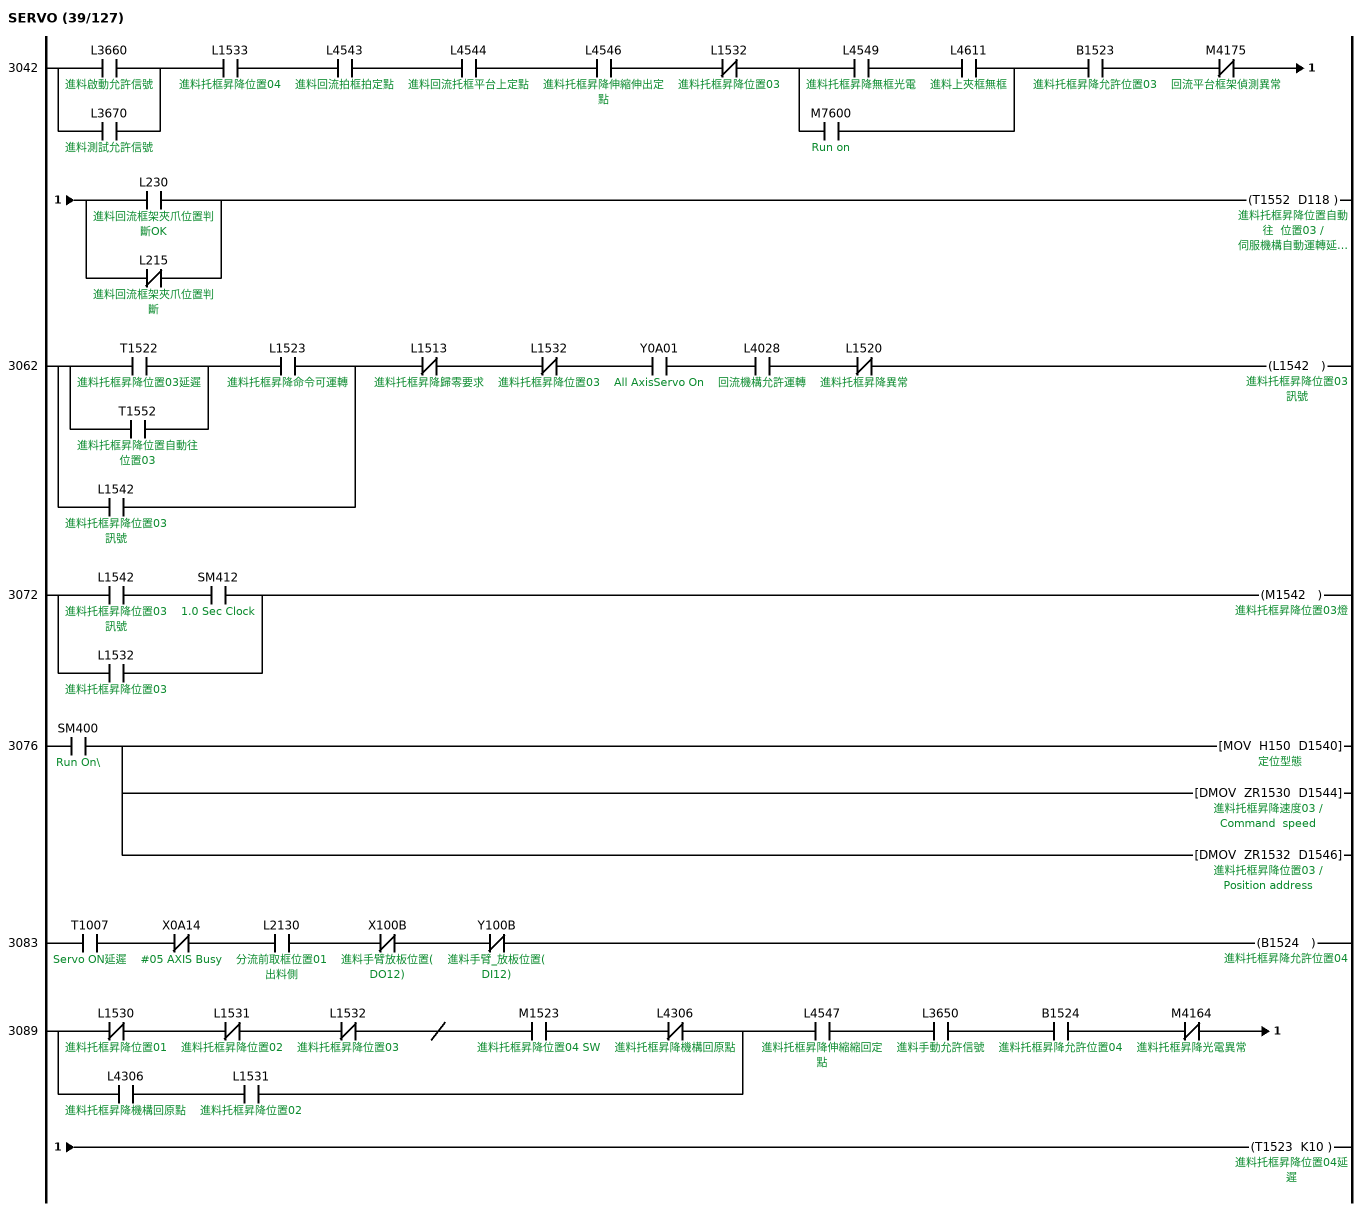
3042  LD      L3660  ; 進料啟動允許信號
      OR      L3670  ; 進料測試允許信號
      AND     L1533  ; 進料托框昇降位置04
      AND     L4543  ; 進料回流拍框拍定點
      AND     L4544  ; 進料回流托框平台上定點
      AND     L4546  ; 進料托框昇降伸縮伸出定點
      ANI     L1532  ; 進料托框昇降位置03
      LD      L4549  ; 進料托框昇降無框光電
      AND     L4611  ; 進料上夾框無框
      OR      M7600  ; Run on
      ANB
      AND     B1523  ; 進料托框昇降允許位置03
      ANI     M4175  ; 回流平台框架偵測異常
      LD      L230  ; 進料回流框架夾爪位置判斷OK
      ORI     L215  ; 進料回流框架夾爪位置判斷
      ANB
      OUT     T1552 D118  ; 進料托框昇降位置自動往  位置03 / 伺服機構自動運轉延遲時間
3062  LD      T1522  ; 進料托框昇降位置03延遲
      OR      T1552  ; 進料托框昇降位置自動往  位置03
      AND     L1523  ; 進料托框昇降命令可運轉
      OR      L1542  ; 進料托框昇降位置03 訊號
      ANI     L1513  ; 進料托框昇降歸零要求
      ANI     L1532  ; 進料托框昇降位置03
      AND     Y0A01  ; All AxisServo On
      AND     L4028  ; 回流機構允許運轉
      ANI     L1520  ; 進料托框昇降異常
      OUT     L1542  ; 進料托框昇降位置03 訊號
3072  LD      L1542  ; 進料托框昇降位置03 訊號
      AND     SM412  ; 1.0 Sec Clock
      OR      L1532  ; 進料托框昇降位置03
      OUT     M1542  ; 進料托框昇降位置03燈
3076  LD      SM400  ; Run On\
      MOV     H150 D1540  ; 定位型態
      DMOV    ZR1530 D1544  ; 進料托框昇降速度03 / Command  speed
      DMOV    ZR1532 D1546  ; Position address
3083  LD      T1007  ; Servo ON延遲
      ANI     X0A14  ; #05 AXIS Busy
      AND     L2130  ; 分流前取框位置01  出料側
      ANI     X100B  ; 進料手臂放板位置(DO12)
      ANI     Y100B  ; 進料手臂_放板位置(DI12)
      OUT     B1524  ; 進料托框昇降允許位置04
3089  LDI     L1530  ; 進料托框昇降位置01
      ANI     L1531  ; 進料托框昇降位置02
      ANI     L1532  ; 進料托框昇降位置03
      INV
      AND     M1523  ; 進料托框昇降位置04 SW
      ANI     L4306  ; 進料托框昇降機構回原點
      LD      L4306  ; 進料托框昇降機構回原點
      AND     L1531  ; 進料托框昇降位置02
      ORB
      AND     L4547  ; 進料托框昇降伸縮縮回定點
      AND     L3650  ; 進料手動允許信號
      AND     B1524  ; 進料托框昇降允許位置04
      ANI     M4164  ; 進料托框昇降光電異常
      OUT     T1523 K10  ; 進料托框昇降位置04延遲
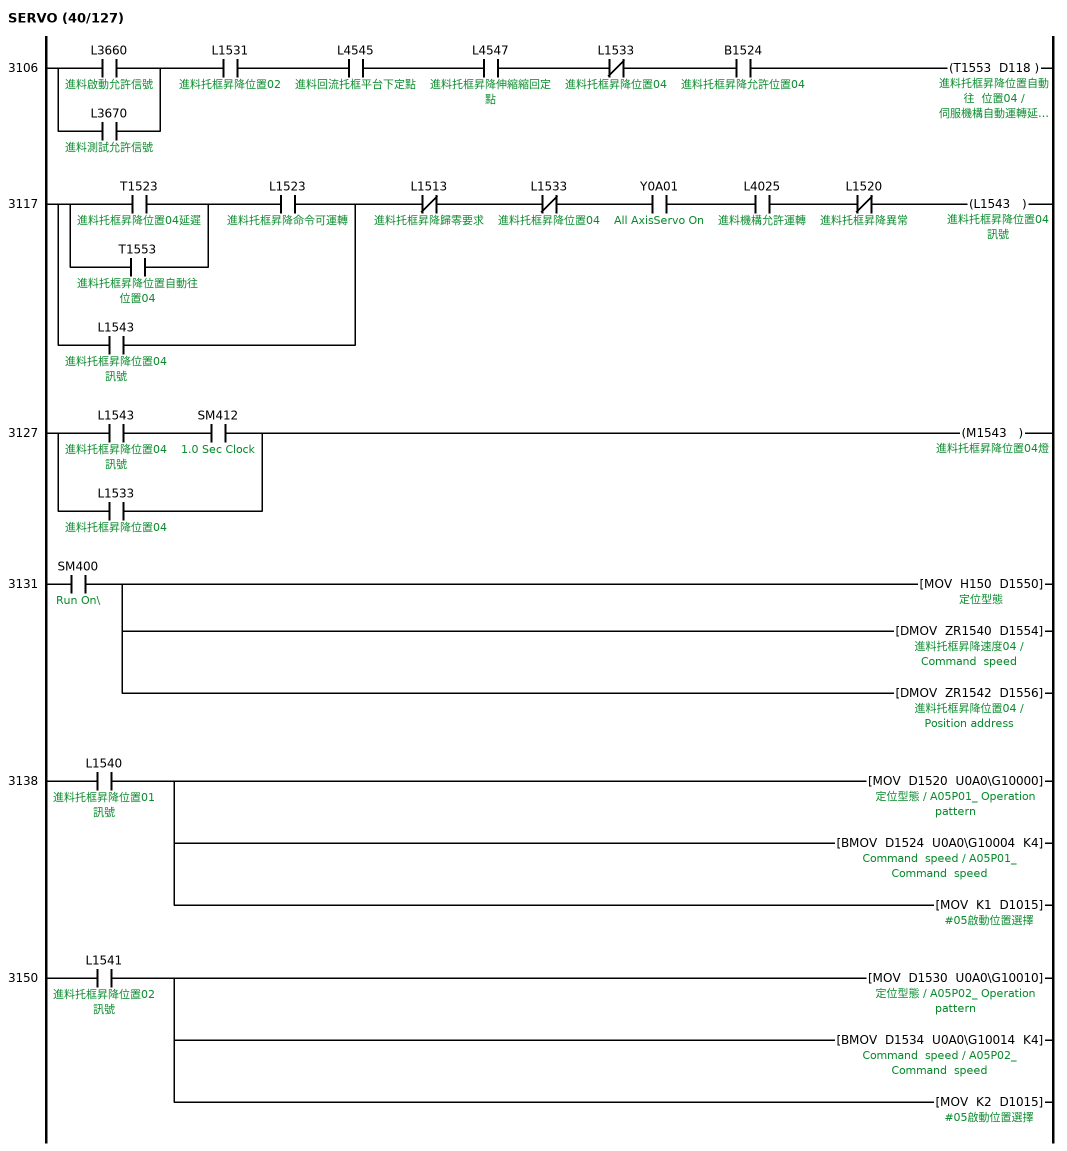
3106  LD      L3660  ; 進料啟動允許信號
      OR      L3670  ; 進料測試允許信號
      AND     L1531  ; 進料托框昇降位置02
      AND     L4545  ; 進料回流托框平台下定點
      AND     L4547  ; 進料托框昇降伸縮縮回定點
      ANI     L1533  ; 進料托框昇降位置04
      AND     B1524  ; 進料托框昇降允許位置04
      OUT     T1553 D118  ; 進料托框昇降位置自動往  位置04 / 伺服機構自動運轉延遲時間
3117  LD      T1523  ; 進料托框昇降位置04延遲
      OR      T1553  ; 進料托框昇降位置自動往  位置04
      AND     L1523  ; 進料托框昇降命令可運轉
      OR      L1543  ; 進料托框昇降位置04 訊號
      ANI     L1513  ; 進料托框昇降歸零要求
      ANI     L1533  ; 進料托框昇降位置04
      AND     Y0A01  ; All AxisServo On
      AND     L4025  ; 進料機構允許運轉
      ANI     L1520  ; 進料托框昇降異常
      OUT     L1543  ; 進料托框昇降位置04 訊號
3127  LD      L1543  ; 進料托框昇降位置04 訊號
      AND     SM412  ; 1.0 Sec Clock
      OR      L1533  ; 進料托框昇降位置04
      OUT     M1543  ; 進料托框昇降位置04燈
3131  LD      SM400  ; Run On\
      MOV     H150 D1550  ; 定位型態
      DMOV    ZR1540 D1554  ; 進料托框昇降速度04 / Command  speed
      DMOV    ZR1542 D1556  ; Position address
3138  LD      L1540  ; 進料托框昇降位置01 訊號
      MOV     D1520 U0A0\G10000  ; A05P01_ Operation pattern
      BMOV    D1524 U0A0\G10004 K4  ; A05P01_ Command  speed
      MOV     K1 D1015  ; #05啟動位置選擇
3150  LD      L1541  ; 進料托框昇降位置02 訊號
      MOV     D1530 U0A0\G10010  ; A05P02_ Operation pattern
      BMOV    D1534 U0A0\G10014 K4  ; A05P02_ Command  speed
      MOV     K2 D1015
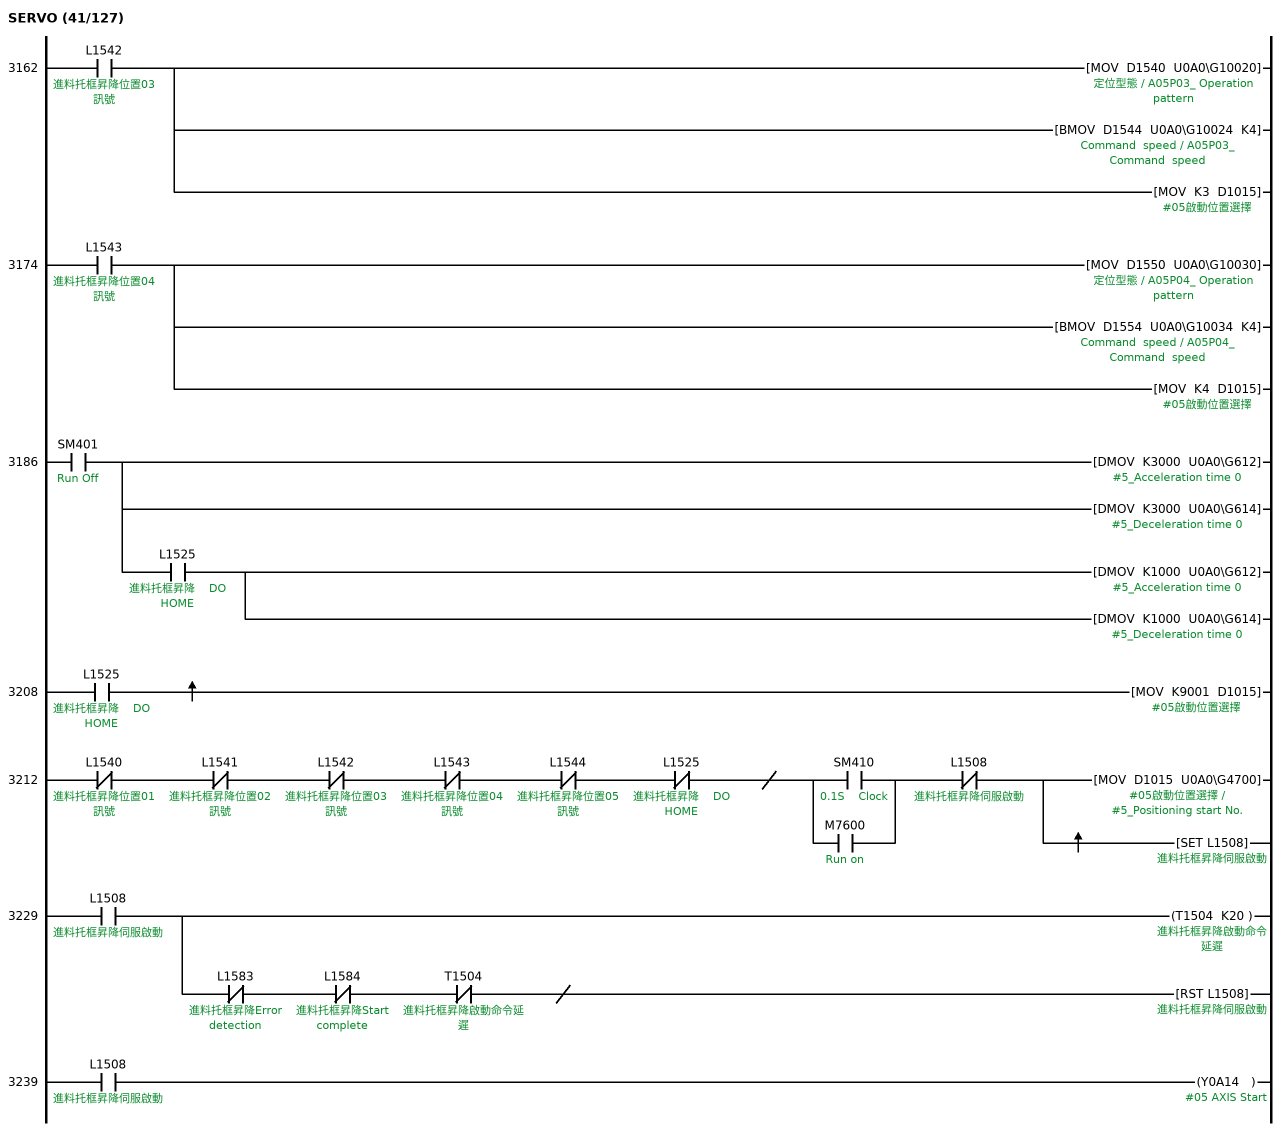
3162  LD      L1542  ; 進料托框昇降位置03 訊號
      MOV     D1540 U0A0\G10020  ; A05P03_ Operation pattern
      BMOV    D1544 U0A0\G10024 K4  ; A05P03_ Command  speed
      MOV     K3 D1015
3174  LD      L1543  ; 進料托框昇降位置04 訊號
      MOV     D1550 U0A0\G10030  ; A05P04_ Operation pattern
      BMOV    D1554 U0A0\G10034 K4  ; A05P04_ Command  speed
      MOV     K4 D1015
3186  LD      SM401  ; Run Off
      DMOV    K3000 U0A0\G612  ; #5_Acceleration time 0
      DMOV    K3000 U0A0\G614  ; #5_Deceleration time 0
      AND     L1525  ; 進料托框昇降    DO HOME
      DMOV    K1000 U0A0\G612
      DMOV    K1000 U0A0\G614
3208  LD      L1525  ; 進料托框昇降    DO HOME
      MEP
      MOV     K9001 D1015
3212  LDI     L1540  ; 進料托框昇降位置01 訊號
      ANI     L1541  ; 進料托框昇降位置02 訊號
      ANI     L1542  ; 進料托框昇降位置03 訊號
      ANI     L1543  ; 進料托框昇降位置04 訊號
      ANI     L1544  ; 進料托框昇降位置05 訊號
      ANI     L1525  ; 進料托框昇降    DO HOME
      INV
      LD      SM410  ; 0.1S    Clock
      OR      M7600  ; Run on
      ANB
      ANI     L1508  ; 進料托框昇降伺服啟動
      MOV     D1015 U0A0\G4700  ; #5_Positioning start No.
      MEP
      SET     L1508  ; 進料托框昇降伺服啟動
3229  LD      L1508  ; 進料托框昇降伺服啟動
      OUT     T1504 K20  ; 進料托框昇降啟動命令延遲
      ANI     L1583  ; 進料托框昇降Error detection
      ANI     L1584  ; 進料托框昇降Start complete
      ANI     T1504  ; 進料托框昇降啟動命令延遲
      INV
      RST     L1508  ; 進料托框昇降伺服啟動
3239  LD      L1508  ; 進料托框昇降伺服啟動
      OUT     Y0A14  ; #05 AXIS Start
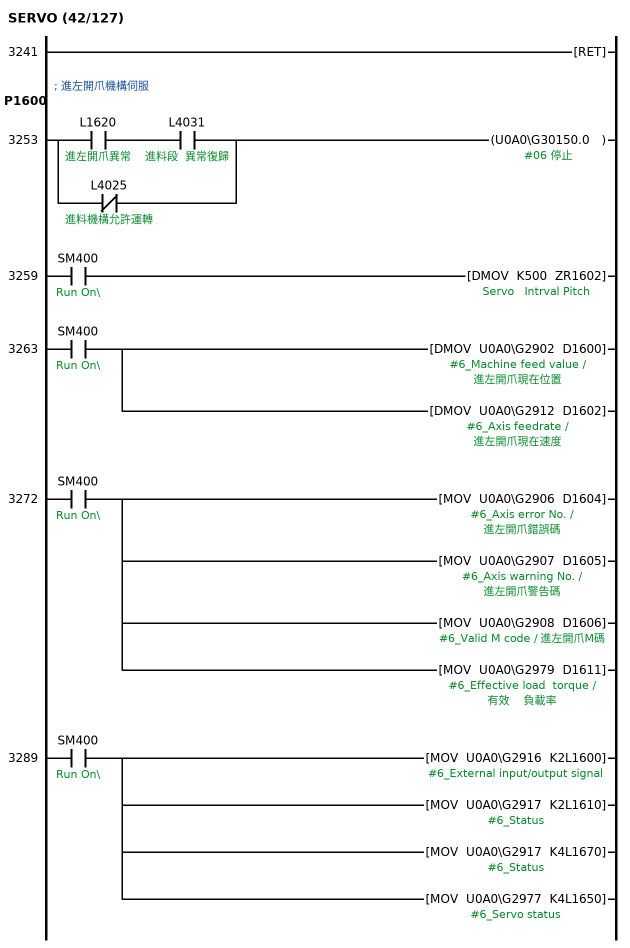
3241  RET
      P1600
; 進左開爪機構伺服
3253  LD      L1620  ; 進左開爪異常
      AND     L4031  ; 進料段  異常復歸
      ORI     L4025  ; 進料機構允許運轉
      OUT     U0A0\G30150.0  ; #06 停止
3259  LD      SM400  ; Run On\
      DMOV    K500 ZR1602  ; Servo   Intrval Pitch
3263  LD      SM400  ; Run On\
      DMOV    U0A0\G2902 D1600  ; #6_Machine feed value / 進左開爪現在位置
      DMOV    U0A0\G2912 D1602  ; #6_Axis feedrate / 進左開爪現在速度
3272  LD      SM400  ; Run On\
      MOV     U0A0\G2906 D1604  ; #6_Axis error No. / 進左開爪錯誤碼
      MOV     U0A0\G2907 D1605  ; #6_Axis warning No. / 進左開爪警告碼
      MOV     U0A0\G2908 D1606  ; #6_Valid M code / 進左開爪M碼
      MOV     U0A0\G2979 D1611  ; #6_Effective load  torque / 有效    負載率
3289  LD      SM400  ; Run On\
      MOV     U0A0\G2916 K2L1600  ; #6_External input/output signal / 進左開爪    負極限
      MOV     U0A0\G2917 K2L1610  ; #6_Status / 進左開爪速度控制
      MOV     U0A0\G2917 K4L1670  ; 進左開爪速度控制
      MOV     U0A0\G2977 K4L1650  ; #6_Servo status / READY ON
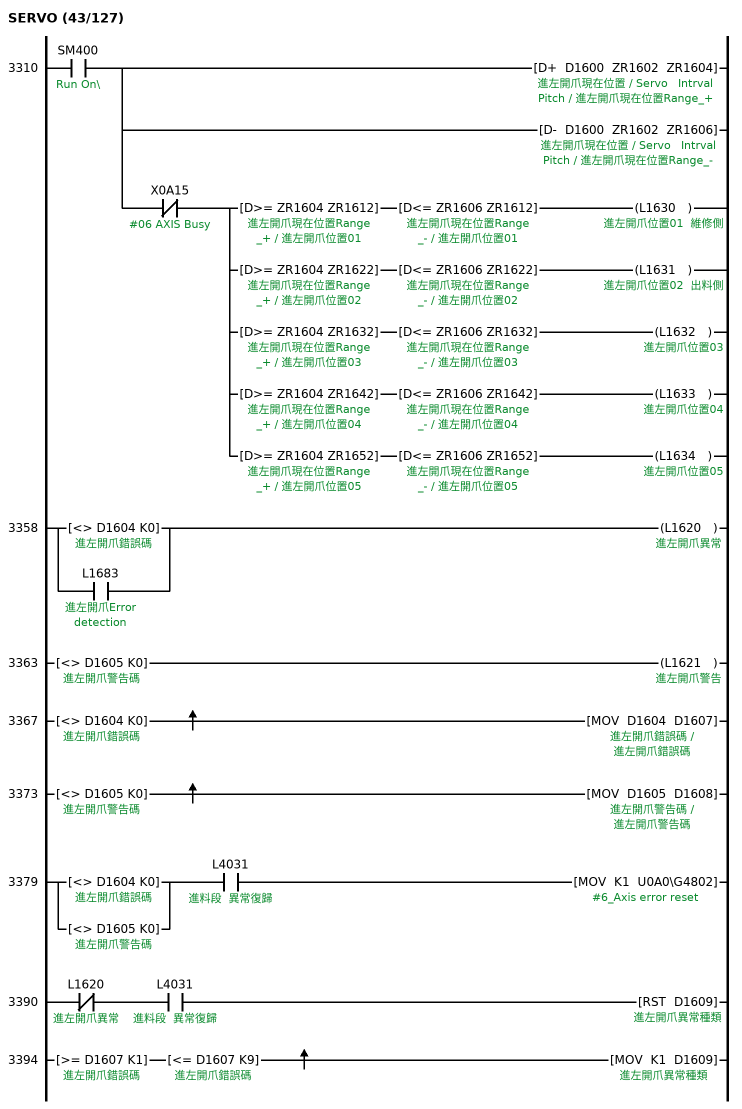
3310  LD      SM400  ; Run On\
      D+      D1600 ZR1602 ZR1604  ; 進左開爪現在位置Range_+
      D-      D1600 ZR1602 ZR1606  ; 進左開爪現在位置Range_-
      ANI     X0A15  ; #06 AXIS Busy
      MPS
      ANDD>=  ZR1604 ZR1612  ; 進左開爪現在位置Range_+ / 進左開爪位置01
      ANDD<=  ZR1606 ZR1612  ; 進左開爪現在位置Range_- / 進左開爪位置01
      OUT     L1630  ; 進左開爪位置01  維修側
      MRD
      ANDD>=  ZR1604 ZR1622  ; 進左開爪現在位置Range_+ / 進左開爪位置02
      ANDD<=  ZR1606 ZR1622  ; 進左開爪現在位置Range_- / 進左開爪位置02
      OUT     L1631  ; 進左開爪位置02  出料側
      MRD
      ANDD>=  ZR1604 ZR1632  ; 進左開爪現在位置Range_+ / 進左開爪位置03
      ANDD<=  ZR1606 ZR1632  ; 進左開爪現在位置Range_- / 進左開爪位置03
      OUT     L1632  ; 進左開爪位置03
      MRD
      ANDD>=  ZR1604 ZR1642  ; 進左開爪現在位置Range_+ / 進左開爪位置04
      ANDD<=  ZR1606 ZR1642  ; 進左開爪現在位置Range_- / 進左開爪位置04
      OUT     L1633  ; 進左開爪位置04
      MPP
      ANDD>=  ZR1604 ZR1652  ; 進左開爪現在位置Range_+ / 進左開爪位置05
      ANDD<=  ZR1606 ZR1652  ; 進左開爪現在位置Range_- / 進左開爪位置05
      OUT     L1634  ; 進左開爪位置05
3358  LD<>    D1604 K0  ; 進左開爪錯誤碼
      OR      L1683  ; 進左開爪Error detection
      OUT     L1620  ; 進左開爪異常
3363  LD<>    D1605 K0  ; 進左開爪警告碼
      OUT     L1621  ; 進左開爪警告
3367  LD<>    D1604 K0  ; 進左開爪錯誤碼
      MEP
      MOV     D1604 D1607  ; 進左開爪錯誤碼
3373  LD<>    D1605 K0  ; 進左開爪警告碼
      MEP
      MOV     D1605 D1608  ; 進左開爪警告碼
3379  LD<>    D1604 K0  ; 進左開爪錯誤碼
      OR<>    D1605 K0  ; 進左開爪警告碼
      AND     L4031  ; 進料段  異常復歸
      MOV     K1 U0A0\G4802  ; #6_Axis error reset
3390  LDI     L1620  ; 進左開爪異常
      AND     L4031  ; 進料段  異常復歸
      RST     D1609  ; 進左開爪異常種類
3394  LD>=    D1607 K1  ; 進左開爪錯誤碼
      AND<=   D1607 K9  ; 進左開爪錯誤碼
      MEP
      MOV     K1 D1609
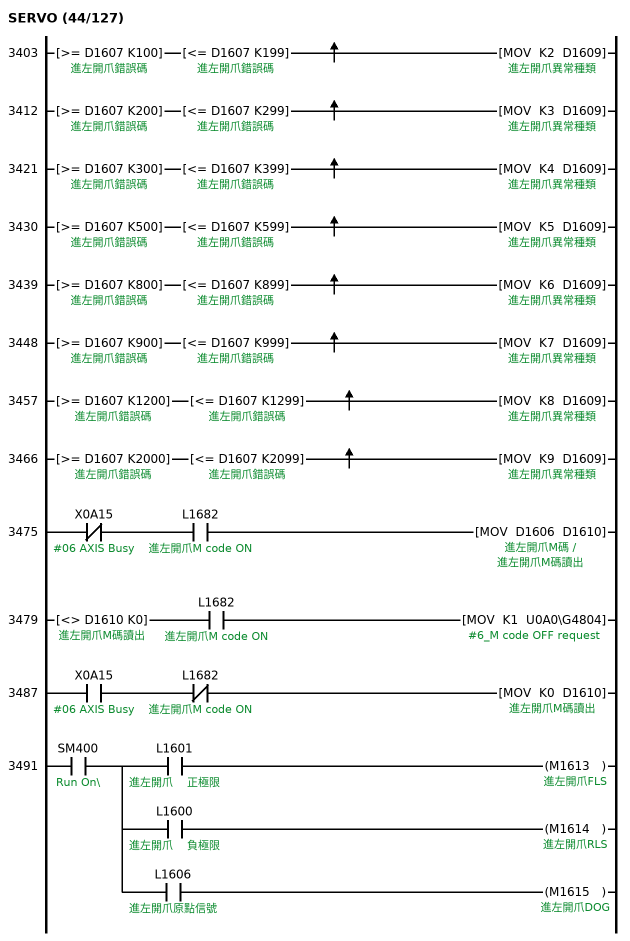
3403  LD>=    D1607 K100  ; 進左開爪錯誤碼
      AND<=   D1607 K199  ; 進左開爪錯誤碼
      MEP
      MOV     K2 D1609
3412  LD>=    D1607 K200  ; 進左開爪錯誤碼
      AND<=   D1607 K299  ; 進左開爪錯誤碼
      MEP
      MOV     K3 D1609
3421  LD>=    D1607 K300  ; 進左開爪錯誤碼
      AND<=   D1607 K399  ; 進左開爪錯誤碼
      MEP
      MOV     K4 D1609
3430  LD>=    D1607 K500  ; 進左開爪錯誤碼
      AND<=   D1607 K599  ; 進左開爪錯誤碼
      MEP
      MOV     K5 D1609
3439  LD>=    D1607 K800  ; 進左開爪錯誤碼
      AND<=   D1607 K899  ; 進左開爪錯誤碼
      MEP
      MOV     K6 D1609
3448  LD>=    D1607 K900  ; 進左開爪錯誤碼
      AND<=   D1607 K999  ; 進左開爪錯誤碼
      MEP
      MOV     K7 D1609
3457  LD>=    D1607 K1200  ; 進左開爪錯誤碼
      AND<=   D1607 K1299  ; 進左開爪錯誤碼
      MEP
      MOV     K8 D1609
3466  LD>=    D1607 K2000  ; 進左開爪錯誤碼
      AND<=   D1607 K2099  ; 進左開爪錯誤碼
      MEP
      MOV     K9 D1609
3475  LDI     X0A15  ; #06 AXIS Busy
      AND     L1682  ; 進左開爪M code ON
      MOV     D1606 D1610  ; 進左開爪M碼讀出
3479  LD<>    D1610 K0  ; 進左開爪M碼讀出
      AND     L1682  ; 進左開爪M code ON
      MOV     K1 U0A0\G4804  ; #6_M code OFF request
3487  LD      X0A15  ; #06 AXIS Busy
      ANI     L1682  ; 進左開爪M code ON
      MOV     K0 D1610
3491  LD      SM400  ; Run On\
      MPS
      AND     L1601  ; 進左開爪    正極限
      OUT     M1613  ; 進左開爪FLS
      MRD
      AND     L1600  ; 進左開爪    負極限
      OUT     M1614  ; 進左開爪RLS
      MPP
      AND     L1606  ; 進左開爪原點信號
      OUT     M1615  ; 進左開爪DOG
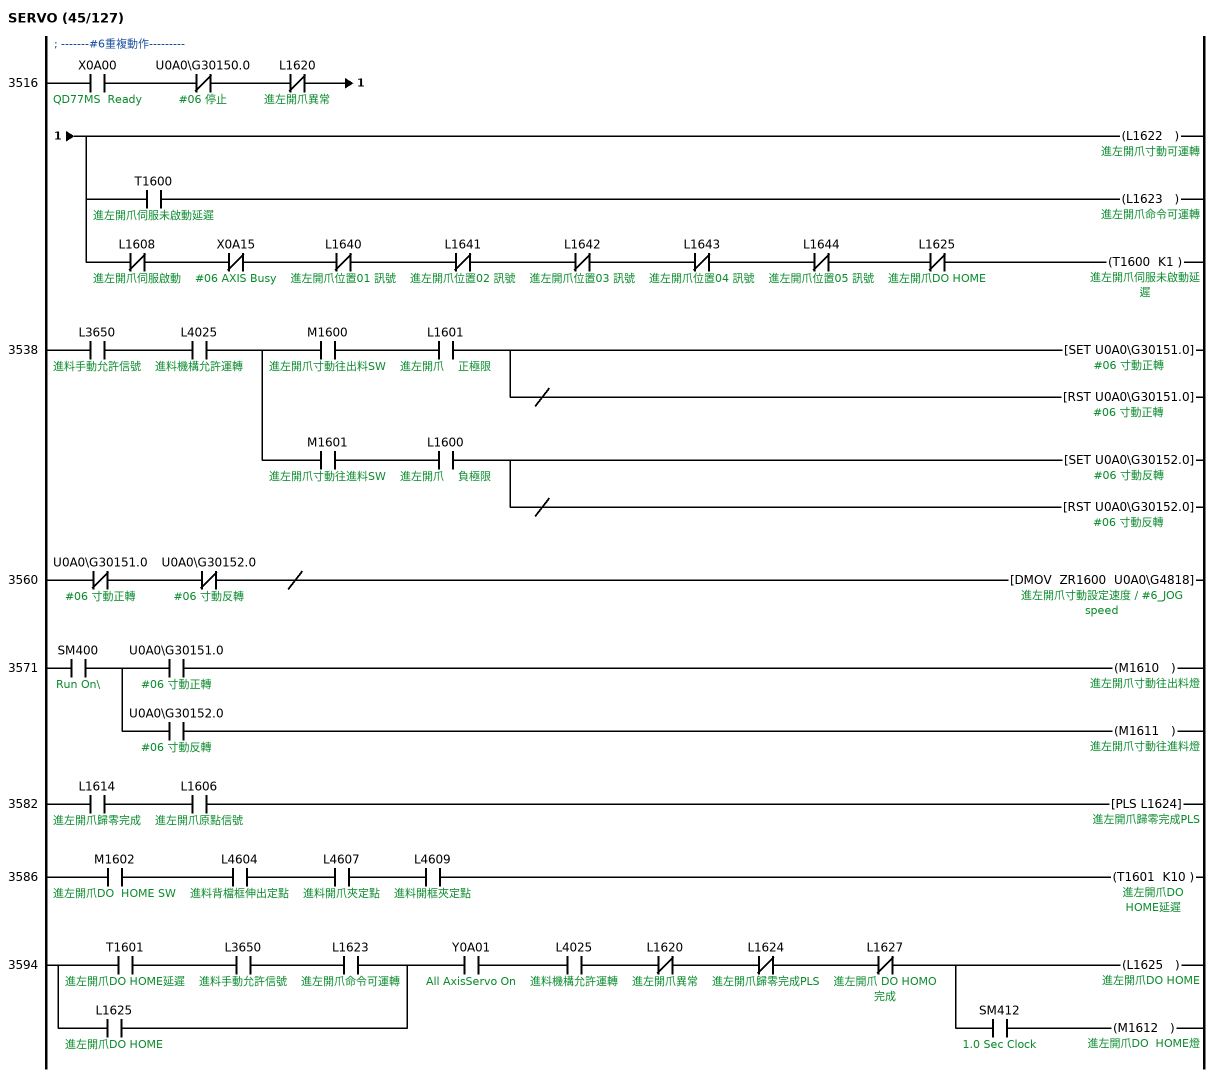
; -------#6重複動作---------
3516  LD      X0A00  ; QD77MS  Ready
      ANI     U0A0\G30150.0  ; #06 停止
      ANI     L1620  ; 進左開爪異常
      OUT     L1622  ; 進左開爪寸動可運轉
      MPS
      AND     T1600  ; 進左開爪伺服未啟動延遲
      OUT     L1623  ; 進左開爪命令可運轉
      MPP
      ANI     L1608  ; 進左開爪伺服啟動
      ANI     X0A15  ; #06 AXIS Busy
      ANI     L1640  ; 進左開爪位置01 訊號
      ANI     L1641  ; 進左開爪位置02 訊號
      ANI     L1642  ; 進左開爪位置03 訊號
      ANI     L1643  ; 進左開爪位置04 訊號
      ANI     L1644  ; 進左開爪位置05 訊號
      ANI     L1625  ; 進左開爪DO HOME
      OUT     T1600 K1  ; 進左開爪伺服未啟動延遲
3538  LD      L3650  ; 進料手動允許信號
      AND     L4025  ; 進料機構允許運轉
      MPS
      AND     M1600  ; 進左開爪寸動往出料SW
      AND     L1601  ; 進左開爪    正極限
      SET     U0A0\G30151.0  ; #06 寸動正轉
      INV
      RST     U0A0\G30151.0  ; #06 寸動正轉
      MPP
      AND     M1601  ; 進左開爪寸動往進料SW
      AND     L1600  ; 進左開爪    負極限
      SET     U0A0\G30152.0  ; #06 寸動反轉
      INV
      RST     U0A0\G30152.0  ; #06 寸動反轉
3560  LDI     U0A0\G30151.0  ; #06 寸動正轉
      ANI     U0A0\G30152.0  ; #06 寸動反轉
      INV
      DMOV    ZR1600 U0A0\G4818  ; 進左開爪寸動設定速度 / #6_JOG     speed
3571  LD      SM400  ; Run On\
      MPS
      AND     U0A0\G30151.0  ; #06 寸動正轉
      OUT     M1610  ; 進左開爪寸動往出料燈
      MPP
      AND     U0A0\G30152.0  ; #06 寸動反轉
      OUT     M1611  ; 進左開爪寸動往進料燈
3582  LD      L1614  ; 進左開爪歸零完成
      AND     L1606  ; 進左開爪原點信號
      PLS     L1624  ; 進左開爪歸零完成PLS
3586  LD      M1602  ; 進左開爪DO  HOME SW
      AND     L4604  ; 進料背檔框伸出定點
      AND     L4607  ; 進料開爪夾定點
      AND     L4609  ; 進料開框夾定點
      OUT     T1601 K10  ; 進左開爪DO HOME延遲
3594  LD      T1601  ; 進左開爪DO HOME延遲
      AND     L3650  ; 進料手動允許信號
      AND     L1623  ; 進左開爪命令可運轉
      OR      L1625  ; 進左開爪DO HOME
      AND     Y0A01  ; All AxisServo On
      AND     L4025  ; 進料機構允許運轉
      ANI     L1620  ; 進左開爪異常
      ANI     L1624  ; 進左開爪歸零完成PLS
      ANI     L1627  ; 進左開爪 DO HOMO 完成
      OUT     L1625  ; 進左開爪DO HOME
      AND     SM412  ; 1.0 Sec Clock
      OUT     M1612  ; 進左開爪DO  HOME燈
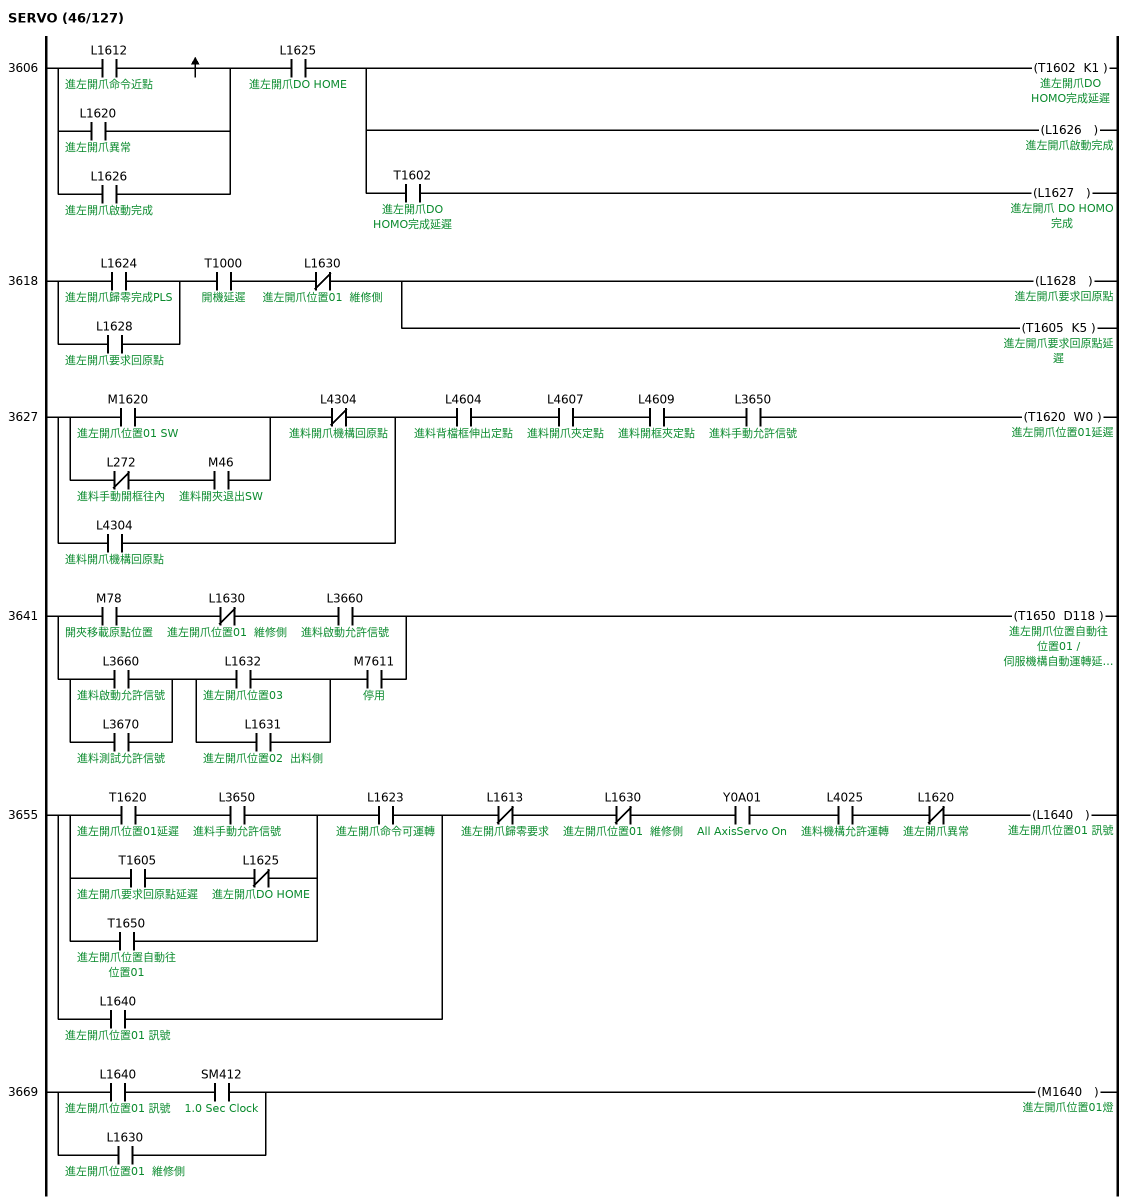
3606  LD      L1612  ; 進左開爪命令近點
      MEP
      OR      L1620  ; 進左開爪異常
      OR      L1626  ; 進左開爪啟動完成
      AND     L1625  ; 進左開爪DO HOME
      OUT     T1602 K1  ; 進左開爪DO HOMO完成延遲
      OUT     L1626  ; 進左開爪啟動完成
      AND     T1602  ; 進左開爪DO HOMO完成延遲
      OUT     L1627  ; 進左開爪 DO HOMO 完成
3618  LD      L1624  ; 進左開爪歸零完成PLS
      OR      L1628  ; 進左開爪要求回原點
      AND     T1000  ; 開機延遲
      ANI     L1630  ; 進左開爪位置01  維修側
      OUT     L1628  ; 進左開爪要求回原點
      OUT     T1605 K5  ; 進左開爪要求回原點延遲
3627  LD      M1620  ; 進左開爪位置01 SW
      LDI     L272  ; 進料手動開框往內
      AND     M46  ; 進料開夾退出SW
      ORB
      ANI     L4304  ; 進料開爪機構回原點
      OR      L4304  ; 進料開爪機構回原點
      AND     L4604  ; 進料背檔框伸出定點
      AND     L4607  ; 進料開爪夾定點
      AND     L4609  ; 進料開框夾定點
      AND     L3650  ; 進料手動允許信號
      OUT     T1620 W0  ; 進左開爪位置01延遲
3641  LD      M78  ; 開夾移載原點位置
      ANI     L1630  ; 進左開爪位置01  維修側
      AND     L3660  ; 進料啟動允許信號
      LD      L3660  ; 進料啟動允許信號
      OR      L3670  ; 進料測試允許信號
      LD      L1632  ; 進左開爪位置03
      OR      L1631  ; 進左開爪位置02  出料側
      ANB
      AND     M7611  ; 停用
      ORB
      OUT     T1650 D118  ; 進左開爪位置自動往  位置01 / 伺服機構自動運轉延遲時間
3655  LD      T1620  ; 進左開爪位置01延遲
      AND     L3650  ; 進料手動允許信號
      LD      T1605  ; 進左開爪要求回原點延遲
      ANI     L1625  ; 進左開爪DO HOME
      ORB
      OR      T1650  ; 進左開爪位置自動往  位置01
      AND     L1623  ; 進左開爪命令可運轉
      OR      L1640  ; 進左開爪位置01 訊號
      ANI     L1613  ; 進左開爪歸零要求
      ANI     L1630  ; 進左開爪位置01  維修側
      AND     Y0A01  ; All AxisServo On
      AND     L4025  ; 進料機構允許運轉
      ANI     L1620  ; 進左開爪異常
      OUT     L1640  ; 進左開爪位置01 訊號
3669  LD      L1640  ; 進左開爪位置01 訊號
      AND     SM412  ; 1.0 Sec Clock
      OR      L1630  ; 進左開爪位置01  維修側
      OUT     M1640  ; 進左開爪位置01燈
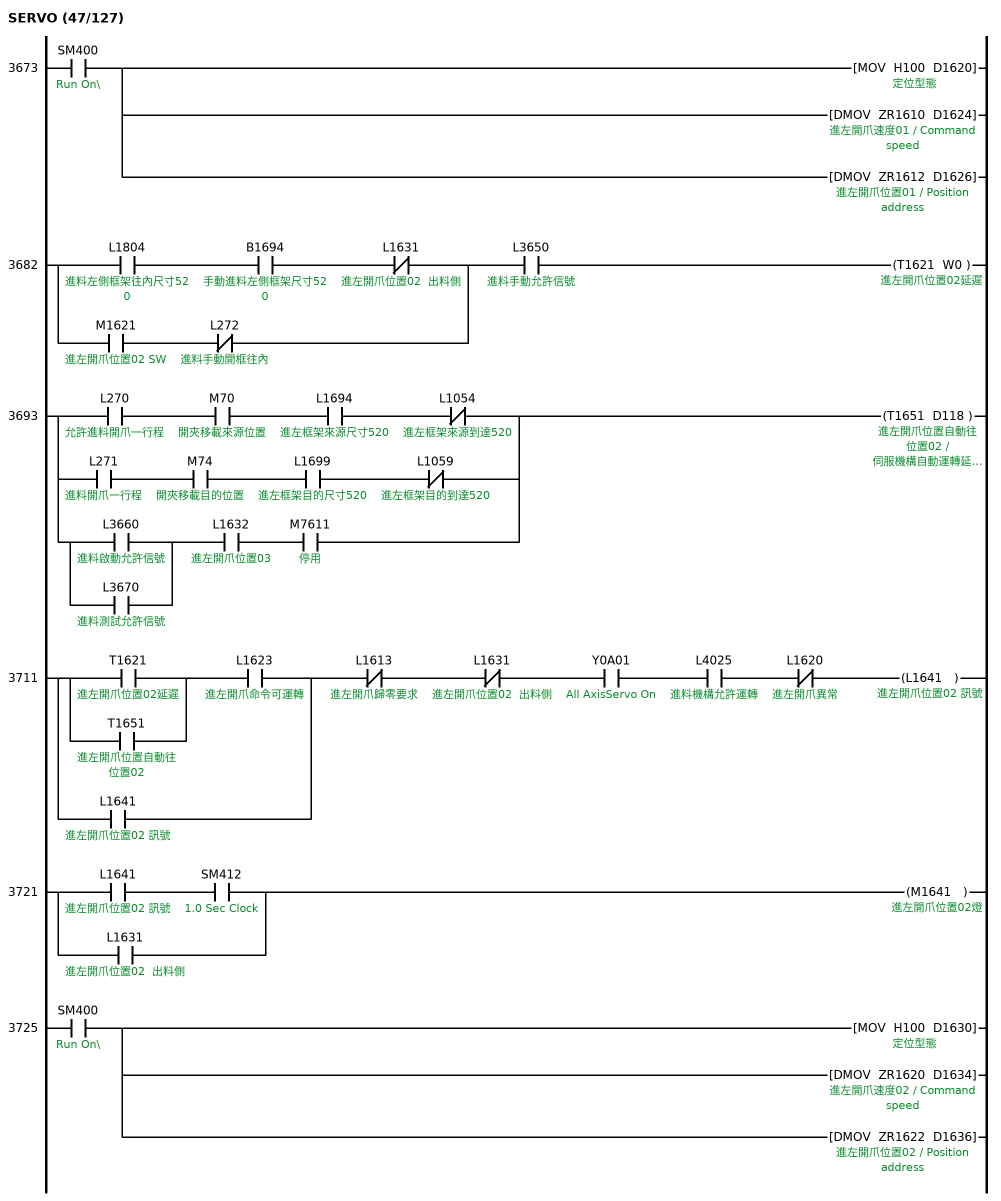
3673  LD      SM400  ; Run On\
      MOV     H100 D1620  ; 定位型態
      DMOV    ZR1610 D1624  ; 進左開爪速度01 / Command  speed
      DMOV    ZR1612 D1626  ; Position address
3682  LD      L1804  ; 進料左側框架往內尺寸520
      AND     B1694  ; 手動進料左側框架尺寸520
      ANI     L1631  ; 進左開爪位置02  出料側
      LD      M1621  ; 進左開爪位置02 SW
      ANI     L272  ; 進料手動開框往內
      ORB
      AND     L3650  ; 進料手動允許信號
      OUT     T1621 W0  ; 進左開爪位置02延遲
3693  LD      L270  ; 允許進料開爪一行程
      AND     M70  ; 開夾移載來源位置
      AND     L1694  ; 進左框架來源尺寸520
      ANI     L1054  ; 進左框架來源到達520
      LD      L271  ; 進料開爪一行程
      AND     M74  ; 開夾移載目的位置
      AND     L1699  ; 進左框架目的尺寸520
      ANI     L1059  ; 進左框架目的到達520
      ORB
      LD      L3660  ; 進料啟動允許信號
      OR      L3670  ; 進料測試允許信號
      AND     L1632  ; 進左開爪位置03
      AND     M7611  ; 停用
      ORB
      OUT     T1651 D118  ; 進左開爪位置自動往  位置02 / 伺服機構自動運轉延遲時間
3711  LD      T1621  ; 進左開爪位置02延遲
      OR      T1651  ; 進左開爪位置自動往  位置02
      AND     L1623  ; 進左開爪命令可運轉
      OR      L1641  ; 進左開爪位置02 訊號
      ANI     L1613  ; 進左開爪歸零要求
      ANI     L1631  ; 進左開爪位置02  出料側
      AND     Y0A01  ; All AxisServo On
      AND     L4025  ; 進料機構允許運轉
      ANI     L1620  ; 進左開爪異常
      OUT     L1641  ; 進左開爪位置02 訊號
3721  LD      L1641  ; 進左開爪位置02 訊號
      AND     SM412  ; 1.0 Sec Clock
      OR      L1631  ; 進左開爪位置02  出料側
      OUT     M1641  ; 進左開爪位置02燈
3725  LD      SM400  ; Run On\
      MOV     H100 D1630  ; 定位型態
      DMOV    ZR1620 D1634  ; 進左開爪速度02 / Command  speed
      DMOV    ZR1622 D1636  ; Position address
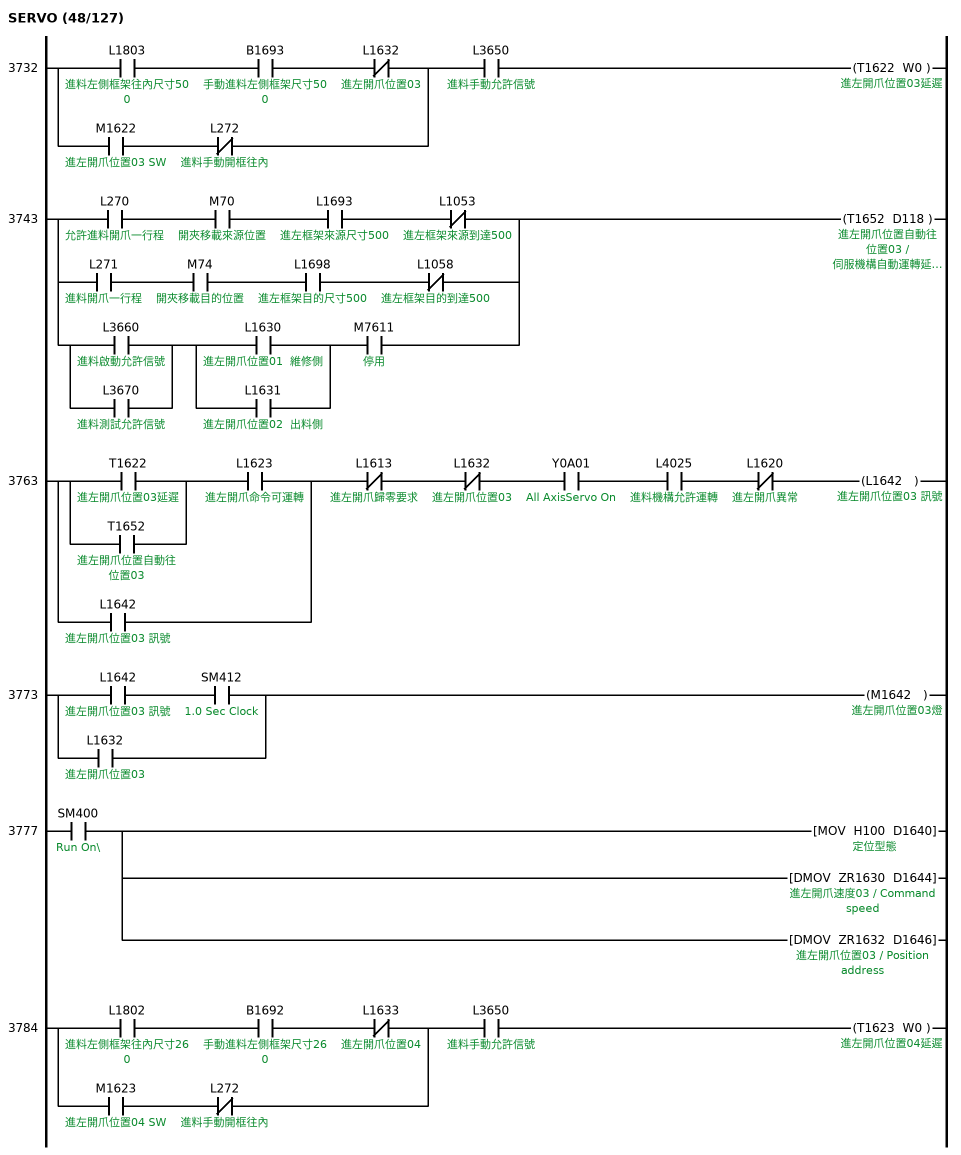
3732  LD      L1803  ; 進料左側框架往內尺寸500
      AND     B1693  ; 手動進料左側框架尺寸500
      ANI     L1632  ; 進左開爪位置03
      LD      M1622  ; 進左開爪位置03 SW
      ANI     L272  ; 進料手動開框往內
      ORB
      AND     L3650  ; 進料手動允許信號
      OUT     T1622 W0  ; 進左開爪位置03延遲
3743  LD      L270  ; 允許進料開爪一行程
      AND     M70  ; 開夾移載來源位置
      AND     L1693  ; 進左框架來源尺寸500
      ANI     L1053  ; 進左框架來源到達500
      LD      L271  ; 進料開爪一行程
      AND     M74  ; 開夾移載目的位置
      AND     L1698  ; 進左框架目的尺寸500
      ANI     L1058  ; 進左框架目的到達500
      ORB
      LD      L3660  ; 進料啟動允許信號
      OR      L3670  ; 進料測試允許信號
      LD      L1630  ; 進左開爪位置01  維修側
      OR      L1631  ; 進左開爪位置02  出料側
      ANB
      AND     M7611  ; 停用
      ORB
      OUT     T1652 D118  ; 進左開爪位置自動往  位置03 / 伺服機構自動運轉延遲時間
3763  LD      T1622  ; 進左開爪位置03延遲
      OR      T1652  ; 進左開爪位置自動往  位置03
      AND     L1623  ; 進左開爪命令可運轉
      OR      L1642  ; 進左開爪位置03 訊號
      ANI     L1613  ; 進左開爪歸零要求
      ANI     L1632  ; 進左開爪位置03
      AND     Y0A01  ; All AxisServo On
      AND     L4025  ; 進料機構允許運轉
      ANI     L1620  ; 進左開爪異常
      OUT     L1642  ; 進左開爪位置03 訊號
3773  LD      L1642  ; 進左開爪位置03 訊號
      AND     SM412  ; 1.0 Sec Clock
      OR      L1632  ; 進左開爪位置03
      OUT     M1642  ; 進左開爪位置03燈
3777  LD      SM400  ; Run On\
      MOV     H100 D1640  ; 定位型態
      DMOV    ZR1630 D1644  ; 進左開爪速度03 / Command  speed
      DMOV    ZR1632 D1646  ; Position address
3784  LD      L1802  ; 進料左側框架往內尺寸260
      AND     B1692  ; 手動進料左側框架尺寸260
      ANI     L1633  ; 進左開爪位置04
      LD      M1623  ; 進左開爪位置04 SW
      ANI     L272  ; 進料手動開框往內
      ORB
      AND     L3650  ; 進料手動允許信號
      OUT     T1623 W0  ; 進左開爪位置04延遲
